LIN {X 0,Y 234.994,Z 198.991,A -85,B 0,C 180,E1 -19665.872,E2 -19665.872} C_VEL
LIN {X 0,Y 235.262,Z 200.964,A -85,B 0,C 180,E1 -19668.915,E2 -19668.915} C_VEL
LIN {X 0,Y 235.336,Z 202.53,A -85,B 0,C 180,E1 -19671.163,E2 -19671.163} C_VEL
LIN {X 0,Y 235.127,Z 205.559,A -85,B 0,C 180,E1 -19675.132,E2 -19675.132} C_VEL
LIN {X 0,Y 236.112,Z 208.531,A -85,B 0,C 180,E1 -19675.455,E2 -19675.455} C_VEL
LIN {X 0,Y 240.672,Z 220.482,A -85,B 0,C 180,E1 -19677.002,E2 -19677.002} C_VEL
LIN {X 0,Y 244.007,Z 232.021,A -85,B 0,C 180,E1 -19678.611,E2 -19678.611} C_VEL
LIN {X 0,Y 246.229,Z 243.079,A -85,B 0,C 180,E1 -19680.305,E2 -19680.305} C_VEL
LIN {X 0,Y 247.437,Z 253.06,A -85,B 0,C 180,E1 -19682.016,E2 -19682.016} C_VEL
LIN {X 0,Y 247.369,Z 256.03,A -85,B 0,C 180,E1 -19682.536,E2 -19682.536} C_VEL
LIN {X 0,Y 245.059,Z 266.116,A -85,B 0,C 180,E1 -19684.294,E2 -19684.294} C_VEL
LIN {X 0,Y 242.891,Z 274.497,A -85,B 0,C 180,E1 -19686.104,E2 -19686.104} C_VEL
LIN {X 0,Y 240.296,Z 283.569,A -85,B 0,C 180,E1 -19688.557,E2 -19688.557} C_VEL
LIN {X 0,Y 238.141,Z 290.868,A -85,B 0,C 180,E1 -19691.057,E2 -19691.057} C_VEL
LIN {X 0,Y 236.506,Z 296.707,A -85,B 0,C 180,E1 -19693.602,E2 -19693.602} C_VEL
LIN {X 0,Y 234.979,Z 301.307,A -85,B 0,C 180,E1 -19696.156,E2 -19696.156} C_VEL
LIN {X 0,Y 234.316,Z 303.742,A -85,B 0,C 180,E1 -19697.88,E2 -19697.88} C_VEL
LIN {X 0,Y 233.756,Z 305.721,A -85,B 0,C 180,E1 -19699.607,E2 -19699.607} C_VEL
LIN {X 0,Y 233.332,Z 307.288,A -85,B 0,C 180,E1 -19701.338,E2 -19701.338} C_VEL
LIN {X 0,Y 233.048,Z 308.446,A -85,B 0,C 180,E1 -19703.071,E2 -19703.071} C_VEL
LIN {X 0,Y 232.884,Z 309.166,A -85,B 0,C 180,E1 -19704.805,E2 -19704.805} C_VEL
LIN {X 0,Y 232.805,Z 309.463,A -85,B 0,C 180,E1 -19708.269,E2 -19708.269} C_VEL
LIN {X 0,Y 232.834,Z 309.041,A -85,B 0,C 180,E1 -19709.999,E2 -19709.999} C_VEL
LIN {X 0,Y 233.162,Z 306.944,A -85,B 0,C 180,E1 -19713.455,E2 -19713.455} C_VEL
LIN {X 0,Y 233.699,Z 304.308,A -85,B 0,C 180,E1 -19716.04,E2 -19716.04} C_VEL
LIN {X 0,Y 234.385,Z 300.675,A -85,B 0,C 180,E1 -19718.621,E2 -19718.621} C_VEL
LIN {X 0,Y 235.457,Z 295.934,A -85,B 0,C 180,E1 -19721.185,E2 -19721.185} C_VEL
LIN {X 0,Y 237.199,Z 288.834,A -85,B 0,C 180,E1 -19724.147,E2 -19724.147} C_VEL
LIN {X 0,Y 239.174,Z 281.069,A -85,B 0,C 180,E1 -19726.646,E2 -19726.646} C_VEL
LIN {X 0,Y 241.478,Z 271.375,A -85,B 0,C 180,E1 -19729.11,E2 -19729.11} C_VEL
LIN {X 0,Y 243.532,Z 261.323,A -85,B 0,C 180,E1 -19731.142,E2 -19731.142} C_VEL
LIN {X 0,Y 245.429,Z 252.166,A -85,B 0,C 180,E1 -19732.608,E2 -19732.608} C_VEL
LIN {X 0,Y 244.466,Z 242.609,A -85,B 0,C 180,E1 -19734.155,E2 -19734.155} C_VEL
LIN {X 0,Y 242.465,Z 231.247,A -85,B 0,C 180,E1 -19735.768,E2 -19735.768} C_VEL
LIN {X 0,Y 239.316,Z 219.271,A -85,B 0,C 180,E1 -19737.274,E2 -19737.274} C_VEL
LIN {X 0,Y 235.407,Z 207.747,A -85,B 0,C 180,E1 -19738.557,E2 -19738.557} C_VEL
LIN {X 0,Y 234.73,Z 205.201,A -85,B 0,C 180,E1 -19738.831,E2 -19738.831} C_VEL
LIN {X 0,Y 235.027,Z 201.864,A -85,B 0,C 180,E1 -19743.144,E2 -19743.144} C_VEL
LIN {X 0,Y 234.981,Z 199.25,A -85,B 0,C 180,E1 -19746.735,E2 -19746.735} C_VEL
LIN {X 0,Y 234.904,Z 198.228,A -85,B 0,C 180,E1 -19748.932,E2 -19748.932} C_VEL
LIN {X 0,Y 234.887,Z 198.229,A -85,B 0,C 180,E1 -19753.481,E2 -19753.481} C_VEL
LIN {X 0,Y 234.963,Z 198.217,A -85,B 0,C 180,E1 -19756.531,E2 -19756.531} C_VEL
LIN {X 0,Y 234.943,Z 198.222,A -85,B 0,C 180,E1 -19761.083,E2 -19761.083} C_VEL
LIN {X 0,Y 234.92,Z 198.222,A -85,B 0,C 180,E1 -19765.36,E2 -19765.36} C_VEL
LIN {X 0,Y 234.906,Z 198.223,A -85,B 0,C 180,E1 -19769.428,E2 -19769.428} C_VEL
LIN {X 0,Y 234.977,Z 198.214,A -85,B 0,C 180,E1 -19773.792,E2 -19773.792} C_VEL
LIN {X 0,Y 235.029,Z 198.172,A -85,B 0,C 180,E1 -19778.971,E2 -19778.971} C_VEL
LIN {X 0,Y 235.098,Z 198.194,A -85,B 0,C 180,E1 -19783.042,E2 -19783.042} C_VEL
LIN {X 0,Y 235.145,Z 198.189,A -85,B 0,C 180,E1 -19787.923,E2 -19787.923} C_VEL
LIN {X 0,Y 235.376,Z 198.162,A -85,B 0,C 180,E1 -19791.414,E2 -19791.414} C_VEL
LIN {X 0,Y 235.388,Z 198.163,A -85,B 0,C 180,E1 -19793.14,E2 -19793.14} C_VEL
LIN {X 0,Y 235.571,Z 198.14,A -85,B 0,C 180,E1 -19798.29,E2 -19798.29} C_VEL
LIN {X 0,Y 235.582,Z 198.14,A -85,B 0,C 180,E1 -19801.709,E2 -19801.709} C_VEL
LIN {X 0,Y 235.381,Z 198.163,A -85,B 0,C 180,E1 -19806.859,E2 -19806.859} C_VEL
LIN {X 0,Y 235.216,Z 198.185,A -85,B 0,C 180,E1 -19810.327,E2 -19810.327} C_VEL
LIN {X 0,Y 235.073,Z 198.205,A -85,B 0,C 180,E1 -19815.609,E2 -19815.609} C_VEL
LIN {X 0,Y 235.009,Z 198.213,A -85,B 0,C 180,E1 -19819.205,E2 -19819.205} C_VEL
LIN {X 0,Y 234.978,Z 198.217,A -85,B 0,C 180,E1 -19822.881,E2 -19822.881} C_VEL
LIN {X 0,Y 234.952,Z 198.219,A -85,B 0,C 180,E1 -19826.659,E2 -19826.659} C_VEL
LIN {X 0,Y 234.914,Z 198.21,A -85,B 0,C 180,E1 -19830.57,E2 -19830.57} C_VEL
LIN {X 0,Y 234.945,Z 198.221,A -85,B 0,C 180,E1 -19834.635,E2 -19834.635} C_VEL
LIN {X 0,Y 234.953,Z 198.219,A -85,B 0,C 180,E1 -19838.955,E2 -19838.955} C_VEL
LIN {X 0,Y 234.997,Z 198.271,A -85,B 0,C 180,E1 -19840.295,E2 -19840.295} C_VEL
LIN {X 0,Y 235.555,Z 201.483,A -85,B 0,C 180,E1 -19844.276,E2 -19844.276} C_VEL
LIN {X 0,Y 236.061,Z 204.807,A -85,B 0,C 180,E1 -19848.099,E2 -19848.099} C_VEL
LIN {X 0,Y 236.491,Z 207.822,A -85,B 0,C 180,E1 -19851.391,E2 -19851.391} C_VEL
LIN {X 0,Y 236.489,Z 209.071,A -85,B 0,C 180,E1 -19852.68,E2 -19852.68} C_VEL
LIN {X 0,Y 235.807,Z 210.061,A -85,B 0,C 180,E1 -19853.591,E2 -19853.591} C_VEL
LIN {X 0,Y 232.815,Z 211.85,A -85,B 0,C 180,E1 -19854.992,E2 -19854.992} C_VEL
LIN {X 0,Y 229.663,Z 213.67,A -85,B 0,C 180,E1 -19856.422,E2 -19856.422} C_VEL
LIN {X 0,Y 228.79,Z 214.713,A -85,B 0,C 180,E1 -19857.371,E2 -19857.371} C_VEL
LIN {X 0,Y 228.579,Z 215.69,A -85,B 0,C 180,E1 -19858.329,E2 -19858.329} C_VEL
LIN {X 0,Y 232.328,Z 229.691,A -85,B 0,C 180,E1 -19859.748,E2 -19859.748} C_VEL
LIN {X 0,Y 234.878,Z 242.527,A -85,B 0,C 180,E1 -19861.279,E2 -19861.279} C_VEL
LIN {X 0,Y 236.253,Z 254.477,A -85,B 0,C 180,E1 -19862.92,E2 -19862.92} C_VEL
LIN {X 0,Y 236.687,Z 265.741,A -85,B 0,C 180,E1 -19864.736,E2 -19864.736} C_VEL
LIN {X 0,Y 236.561,Z 270.846,A -85,B 0,C 180,E1 -19865.659,E2 -19865.659} C_VEL
LIN {X 0,Y 234.302,Z 280.591,A -85,B 0,C 180,E1 -19867.518,E2 -19867.518} C_VEL
LIN {X 0,Y 232.039,Z 290.368,A -85,B 0,C 180,E1 -19869.872,E2 -19869.872} C_VEL
LIN {X 0,Y 230.139,Z 298.132,A -85,B 0,C 180,E1 -19872.221,E2 -19872.221} C_VEL
LIN {X 0,Y 228.441,Z 305.049,A -85,B 0,C 180,E1 -19874.843,E2 -19874.843} C_VEL
LIN {X 0,Y 227.127,Z 310.591,A -85,B 0,C 180,E1 -19877.493,E2 -19877.493} C_VEL
LIN {X 0,Y 226.317,Z 314.942,A -85,B 0,C 180,E1 -19880.168,E2 -19880.168} C_VEL
LIN {X 0,Y 225.82,Z 318.217,A -85,B 0,C 180,E1 -19882.851,E2 -19882.851} C_VEL
LIN {X 0,Y 225.589,Z 320.491,A -85,B 0,C 180,E1 -19885.508,E2 -19885.508} C_VEL
LIN {X 0,Y 225.643,Z 321.872,A -85,B 0,C 180,E1 -19888.216,E2 -19888.216} C_VEL
LIN {X 0,Y 225.714,Z 322.254,A -85,B 0,C 180,E1 -19890.001,E2 -19890.001} C_VEL
LIN {X 0,Y 225.636,Z 322.245,A -85,B 0,C 180,E1 -19891.786,E2 -19891.786} C_VEL
LIN {X 0,Y 225.585,Z 321.472,A -85,B 0,C 180,E1 -19894.48,E2 -19894.48} C_VEL
LIN {X 0,Y 225.822,Z 319.809,A -85,B 0,C 180,E1 -19897.152,E2 -19897.152} C_VEL
LIN {X 0,Y 226.356,Z 317.2,A -85,B 0,C 180,E1 -19899.833,E2 -19899.833} C_VEL
LIN {X 0,Y 227.26,Z 313.584,A -85,B 0,C 180,E1 -19902.502,E2 -19902.502} C_VEL
LIN {X 0,Y 228.572,Z 308.866,A -85,B 0,C 180,E1 -19905.15,E2 -19905.15} C_VEL
LIN {X 0,Y 230.423,Z 302.906,A -85,B 0,C 180,E1 -19907.758,E2 -19907.758} C_VEL
LIN {X 0,Y 232.584,Z 295.571,A -85,B 0,C 180,E1 -19910.305,E2 -19910.305} C_VEL
LIN {X 0,Y 234.7,Z 287.935,A -85,B 0,C 180,E1 -19912.444,E2 -19912.444} C_VEL
LIN {X 0,Y 237.272,Z 278.802,A -85,B 0,C 180,E1 -19914.499,E2 -19914.499} C_VEL
LIN {X 0,Y 238.862,Z 272.268,A -85,B 0,C 180,E1 -19915.72,E2 -19915.72} C_VEL
LIN {X 0,Y 238.703,Z 261.301,A -85,B 0,C 180,E1 -19917.736,E2 -19917.736} C_VEL
LIN {X 0,Y 237.746,Z 250.445,A -85,B 0,C 180,E1 -19919.471,E2 -19919.471} C_VEL
LIN {X 0,Y 235.848,Z 239.193,A -85,B 0,C 180,E1 -19921.074,E2 -19921.074} C_VEL
LIN {X 0,Y 232.84,Z 226.637,A -85,B 0,C 180,E1 -19922.652,E2 -19922.652} C_VEL
LIN {X 0,Y 229.491,Z 216.356,A -85,B 0,C 180,E1 -19923.854,E2 -19923.854} C_VEL
LIN {X 0,Y 229.383,Z 215.464,A -85,B 0,C 180,E1 -19923.937,E2 -19923.937} C_VEL
LIN {X 0,Y 229.656,Z 213.876,A -85,B 0,C 180,E1 -19925.551,E2 -19925.551} C_VEL
LIN {X 0,Y 229.77,Z 210.838,A -85,B 0,C 180,E1 -19928.83,E2 -19928.83} C_VEL
LIN {X 0,Y 229.352,Z 207.534,A -85,B 0,C 180,E1 -19932.657,E2 -19932.657} C_VEL
LIN {X 0,Y 228.983,Z 205.536,A -85,B 0,C 180,E1 -19935.096,E2 -19935.096} C_VEL
LIN {X 0,Y 228.349,Z 202.015,A -85,B 0,C 180,E1 -19939.735,E2 -19939.735} C_VEL
LIN {X 0,Y 227.903,Z 199.162,A -85,B 0,C 180,E1 -19943.813,E2 -19943.813} C_VEL
LIN {X 0,Y 227.848,Z 199.108,A -85,B 0,C 180,E1 -19948.375,E2 -19948.375} C_VEL
LIN {X 0,Y 227.86,Z 199.103,A -85,B 0,C 180,E1 -19952.442,E2 -19952.442} C_VEL
LIN {X 0,Y 227.924,Z 199.094,A -85,B 0,C 180,E1 -19956.369,E2 -19956.369} C_VEL
LIN {X 0,Y 227.957,Z 199.09,A -85,B 0,C 180,E1 -19960.176,E2 -19960.176} C_VEL
LIN {X 0,Y 228.052,Z 199.077,A -85,B 0,C 180,E1 -19963.898,E2 -19963.898} C_VEL
LIN {X 0,Y 228.058,Z 199.075,A -85,B 0,C 180,E1 -19967.543,E2 -19967.543} C_VEL
LIN {X 0,Y 228.255,Z 199.052,A -85,B 0,C 180,E1 -19971.144,E2 -19971.144} C_VEL
LIN {X 0,Y 228.311,Z 199.046,A -85,B 0,C 180,E1 -19972.928,E2 -19972.928} C_VEL
LIN {X 0,Y 228.538,Z 199.017,A -85,B 0,C 180,E1 -19978.238,E2 -19978.238} C_VEL
LIN {X 0,Y 228.551,Z 199.015,A -85,B 0,C 180,E1 -19981.763,E2 -19981.763} C_VEL
LIN {X 0,Y 228.308,Z 199.044,A -85,B 0,C 180,E1 -19987.073,E2 -19987.073} C_VEL
LIN {X 0,Y 228.13,Z 199.067,A -85,B 0,C 180,E1 -19990.652,E2 -19990.652} C_VEL
LIN {X 0,Y 228.04,Z 199.079,A -85,B 0,C 180,E1 -19996.104,E2 -19996.104} C_VEL
LIN {X 0,Y 227.931,Z 199.093,A -85,B 0,C 180,E1 -19999.827,E2 -19999.827} C_VEL
LIN {X 0,Y 227.904,Z 199.096,A -85,B 0,C 180,E1 -20003.634,E2 -20003.634} C_VEL
LIN {X 0,Y 227.871,Z 199.101,A -85,B 0,C 180,E1 -20007.558,E2 -20007.558} C_VEL
LIN {X 0,Y 227.859,Z 199.102,A -85,B 0,C 180,E1 -20011.625,E2 -20011.625} C_VEL
LIN {X 0,Y 227.875,Z 199.1,A -85,B 0,C 180,E1 -20015.874,E2 -20015.874} C_VEL
LIN {X 0,Y 227.82,Z 199.106,A -85,B 0,C 180,E1 -20020.379,E2 -20020.379} C_VEL
LIN {X 0,Y 227.8,Z 199.111,A -85,B 0,C 180,E1 -20022.746,E2 -20022.746} C_VEL
LIN {X 0,Y 227.93,Z 199.817,A -85,B 0,C 180,E1 -20025.169,E2 -20025.169} C_VEL
LIN {X 0,Y 228.262,Z 202.698,A -85,B 0,C 180,E1 -20029.718,E2 -20029.718} C_VEL
LIN {X 0,Y 228.207,Z 205.665,A -85,B 0,C 180,E1 -20033.954,E2 -20033.954} C_VEL
LIN {X 0,Y 229.317,Z 208.854,A -85,B 0,C 180,E1 -20034.329,E2 -20034.329} C_VEL
LIN {X 0,Y 233.879,Z 220.739,A -85,B 0,C 180,E1 -20035.961,E2 -20035.961} C_VEL
LIN {X 0,Y 236.893,Z 230.669,A -85,B 0,C 180,E1 -20037.423,E2 -20037.423} C_VEL
LIN {X 0,Y 239.325,Z 241.897,A -85,B 0,C 180,E1 -20039.201,E2 -20039.201} C_VEL
LIN {X 0,Y 240.688,Z 251.922,A -85,B 0,C 180,E1 -20040.963,E2 -20040.963} C_VEL
LIN {X 0,Y 240.842,Z 257.166,A -85,B 0,C 180,E1 -20041.934,E2 -20041.934} C_VEL
LIN {X 0,Y 238.38,Z 267.157,A -85,B 0,C 180,E1 -20043.754,E2 -20043.754} C_VEL
LIN {X 0,Y 235.922,Z 276.204,A -85,B 0,C 180,E1 -20045.821,E2 -20045.821} C_VEL
LIN {X 0,Y 233.255,Z 285.017,A -85,B 0,C 180,E1 -20048.341,E2 -20048.341} C_VEL
LIN {X 0,Y 231.074,Z 292.072,A -85,B 0,C 180,E1 -20050.916,E2 -20050.916} C_VEL
LIN {X 0,Y 229.676,Z 296.838,A -85,B 0,C 180,E1 -20053.1,E2 -20053.1} C_VEL
LIN {X 0,Y 228.059,Z 301.452,A -85,B 0,C 180,E1 -20055.727,E2 -20055.727} C_VEL
LIN {X 0,Y 227.355,Z 303.901,A -85,B 0,C 180,E1 -20057.503,E2 -20057.503} C_VEL
LIN {X 0,Y 226.758,Z 305.886,A -85,B 0,C 180,E1 -20059.282,E2 -20059.282} C_VEL
LIN {X 0,Y 226.293,Z 307.46,A -85,B 0,C 180,E1 -20061.066,E2 -20061.066} C_VEL
LIN {X 0,Y 225.996,Z 308.626,A -85,B 0,C 180,E1 -20062.854,E2 -20062.854} C_VEL
LIN {X 0,Y 225.768,Z 309.442,A -85,B 0,C 180,E1 -20064.972,E2 -20064.972} C_VEL
LIN {X 0,Y 225.72,Z 309.664,A -85,B 0,C 180,E1 -20068.215,E2 -20068.215} C_VEL
LIN {X 0,Y 225.747,Z 309.25,A -85,B 0,C 180,E1 -20069.999,E2 -20069.999} C_VEL
LIN {X 0,Y 225.853,Z 308.408,A -85,B 0,C 180,E1 -20071.782,E2 -20071.782} C_VEL
LIN {X 0,Y 226.09,Z 307.168,A -85,B 0,C 180,E1 -20073.563,E2 -20073.563} C_VEL
LIN {X 0,Y 226.634,Z 304.545,A -85,B 0,C 180,E1 -20076.229,E2 -20076.229} C_VEL
LIN {X 0,Y 227.379,Z 300.925,A -85,B 0,C 180,E1 -20078.888,E2 -20078.888} C_VEL
LIN {X 0,Y 228.519,Z 296.198,A -85,B 0,C 180,E1 -20081.529,E2 -20081.529} C_VEL
LIN {X 0,Y 230.331,Z 289.114,A -85,B 0,C 180,E1 -20084.578,E2 -20084.578} C_VEL
LIN {X 0,Y 232.401,Z 281.376,A -85,B 0,C 180,E1 -20087.146,E2 -20087.146} C_VEL
LIN {X 0,Y 234.778,Z 271.705,A -85,B 0,C 180,E1 -20089.677,E2 -20089.677} C_VEL
LIN {X 0,Y 236.948,Z 261.692,A -85,B 0,C 180,E1 -20091.759,E2 -20091.759} C_VEL
LIN {X 0,Y 238.789,Z 253.116,A -85,B 0,C 180,E1 -20093.18,E2 -20093.18} C_VEL
LIN {X 0,Y 237.942,Z 244.186,A -85,B 0,C 180,E1 -20094.695,E2 -20094.695} C_VEL
LIN {X 0,Y 236.166,Z 233.622,A -85,B 0,C 180,E1 -20096.299,E2 -20096.299} C_VEL
LIN {X 0,Y 233.467,Z 222.697,A -85,B 0,C 180,E1 -20097.782,E2 -20097.782} C_VEL
LIN {X 0,Y 229.335,Z 210.086,A -85,B 0,C 180,E1 -20099.303,E2 -20099.303} C_VEL
LIN {X 0,Y 227.736,Z 205.422,A -85,B 0,C 180,E1 -20099.839,E2 -20099.839} C_VEL
LIN {X 0,Y 228.003,Z 202.525,A -85,B 0,C 180,E1 -20103.695,E2 -20103.695} C_VEL
LIN {X 0,Y 227.982,Z 200.413,A -85,B 0,C 180,E1 -20106.725,E2 -20106.725} C_VEL
LIN {X 0,Y 227.856,Z 199.502,A -85,B 0,C 180,E1 -20108.084,E2 -20108.084} C_VEL
LIN {X 0,Y 227.811,Z 199.109,A -85,B 0,C 180,E1 -20110.375,E2 -20110.375} C_VEL
LIN {X 0,Y 227.85,Z 199.103,A -85,B 0,C 180,E1 -20115.183,E2 -20115.183} C_VEL
LIN {X 0,Y 227.906,Z 199.097,A -85,B 0,C 180,E1 -20117.733,E2 -20117.733} C_VEL
LIN {X 0,Y 227.856,Z 199.101,A -85,B 0,C 180,E1 -20121.91,E2 -20121.91} C_VEL
LIN {X 0,Y 227.866,Z 199.101,A -85,B 0,C 180,E1 -20126.374,E2 -20126.374} C_VEL
LIN {X 0,Y 227.888,Z 199.098,A -85,B 0,C 180,E1 -20130.433,E2 -20130.433} C_VEL
LIN {X 0,Y 227.914,Z 199.093,A -85,B 0,C 180,E1 -20134.423,E2 -20134.423} C_VEL
LIN {X 0,Y 227.99,Z 199.05,A -85,B 0,C 180,E1 -20138.289,E2 -20138.289} C_VEL
LIN {X 0,Y 228.026,Z 199.071,A -85,B 0,C 180,E1 -20142.816,E2 -20142.816} C_VEL
LIN {X 0,Y 228.086,Z 199.071,A -85,B 0,C 180,E1 -20147.543,E2 -20147.543} C_VEL
LIN {X 0,Y 228.314,Z 199.041,A -85,B 0,C 180,E1 -20151.146,E2 -20151.146} C_VEL
LIN {X 0,Y 228.341,Z 199.04,A -85,B 0,C 180,E1 -20152.928,E2 -20152.928} C_VEL
LIN {X 0,Y 228.53,Z 199.017,A -85,B 0,C 180,E1 -20158.237,E2 -20158.237} C_VEL
LIN {X 0,Y 228.542,Z 199.017,A -85,B 0,C 180,E1 -20161.762,E2 -20161.762} C_VEL
LIN {X 0,Y 228.332,Z 199.042,A -85,B 0,C 180,E1 -20167.072,E2 -20167.072} C_VEL
LIN {X 0,Y 228.137,Z 199.067,A -85,B 0,C 180,E1 -20170.651,E2 -20170.651} C_VEL
LIN {X 0,Y 228.024,Z 199.081,A -85,B 0,C 180,E1 -20176.104,E2 -20176.104} C_VEL
LIN {X 0,Y 227.947,Z 199.092,A -85,B 0,C 180,E1 -20179.825,E2 -20179.825} C_VEL
LIN {X 0,Y 227.916,Z 199.095,A -85,B 0,C 180,E1 -20183.632,E2 -20183.632} C_VEL
LIN {X 0,Y 227.868,Z 199.1,A -85,B 0,C 180,E1 -20187.557,E2 -20187.557} C_VEL
LIN {X 0,Y 227.856,Z 199.092,A -85,B 0,C 180,E1 -20191.624,E2 -20191.624} C_VEL
LIN {X 0,Y 227.886,Z 199.099,A -85,B 0,C 180,E1 -20195.871,E2 -20195.871} C_VEL
LIN {X 0,Y 227.988,Z 199.297,A -85,B 0,C 180,E1 -20199.876,E2 -20199.876} C_VEL
LIN {X 0,Y 228.357,Z 201.395,A -85,B 0,C 180,E1 -20202.616,E2 -20202.616} C_VEL
LIN {X 0,Y 228.977,Z 205.386,A -85,B 0,C 180,E1 -20207.445,E2 -20207.445} C_VEL
LIN {X 0,Y 229.444,Z 208.657,A -85,B 0,C 180,E1 -20211.143,E2 -20211.143} C_VEL
LIN {X 0,Y 229.38,Z 211.736,A -85,B 0,C 180,E1 -20214.403,E2 -20214.403} C_VEL
LIN {X 0,Y 228.79,Z 214.713,A -85,B 0,C 180,E1 -20217.371,E2 -20217.371} C_VEL
LIN {X 0,Y 229.046,Z 215.928,A -85,B 0,C 180,E1 -20218.009,E2 -20218.009} C_VEL
LIN {X 0,Y 230.107,Z 218.575,A -85,B 0,C 180,E1 -20218.663,E2 -20218.663} C_VEL
LIN {X 0,Y 231.77,Z 222.871,A -85,B 0,C 180,E1 -20219.187,E2 -20219.187} C_VEL
LIN {X 0,Y 232.069,Z 226.734,A -85,B 0,C 180,E1 -20219.491,E2 -20219.491} C_VEL
LIN {X 0,Y 231.275,Z 231.15,A -85,B 0,C 180,E1 -20219.698,E2 -20219.698} C_VEL
LIN {X 0,Y 228.54,Z 239.929,A -85,B 0,C 180,E1 -20220.171,E2 -20220.171} C_VEL
LIN {X 0,Y 228.37,Z 243.73,A -85,B 0,C 180,E1 -20220.571,E2 -20220.571} C_VEL
LIN {X 0,Y 229.614,Z 254.399,A -85,B 0,C 180,E1 -20222.121,E2 -20222.121} C_VEL
LIN {X 0,Y 229.988,Z 265.661,A -85,B 0,C 180,E1 -20224.002,E2 -20224.002} C_VEL
LIN {X 0,Y 229.823,Z 271.676,A -85,B 0,C 180,E1 -20225.139,E2 -20225.139} C_VEL
LIN {X 0,Y 227.265,Z 282.226,A -85,B 0,C 180,E1 -20227.263,E2 -20227.263} C_VEL
LIN {X 0,Y 225.196,Z 290.719,A -85,B 0,C 180,E1 -20229.431,E2 -20229.431} C_VEL
LIN {X 0,Y 223.37,Z 297.855,A -85,B 0,C 180,E1 -20231.664,E2 -20231.664} C_VEL
LIN {X 0,Y 221.57,Z 304.786,A -85,B 0,C 180,E1 -20234.361,E2 -20234.361} C_VEL
LIN {X 0,Y 220.144,Z 310.34,A -85,B 0,C 180,E1 -20237.089,E2 -20237.089} C_VEL
LIN {X 0,Y 219.301,Z 314.704,A -85,B 0,C 180,E1 -20239.85,E2 -20239.85} C_VEL
LIN {X 0,Y 218.759,Z 317.99,A -85,B 0,C 180,E1 -20242.618,E2 -20242.618} C_VEL
LIN {X 0,Y 218.486,Z 320.475,A -85,B 0,C 180,E1 -20245.688,E2 -20245.688} C_VEL
LIN {X 0,Y 218.541,Z 321.666,A -85,B 0,C 180,E1 -20248.159,E2 -20248.159} C_VEL
LIN {X 0,Y 218.629,Z 322.054,A -85,B 0,C 180,E1 -20250.001,E2 -20250.001} C_VEL
LIN {X 0,Y 218.534,Z 322.05,A -85,B 0,C 180,E1 -20251.844,E2 -20251.844} C_VEL
LIN {X 0,Y 218.482,Z 321.432,A -85,B 0,C 180,E1 -20254.297,E2 -20254.297} C_VEL
LIN {X 0,Y 218.761,Z 319.634,A -85,B 0,C 180,E1 -20257.384,E2 -20257.384} C_VEL
LIN {X 0,Y 219.339,Z 317.036,A -85,B 0,C 180,E1 -20260.151,E2 -20260.151} C_VEL
LIN {X 0,Y 220.28,Z 313.43,A -85,B 0,C 180,E1 -20262.905,E2 -20262.905} C_VEL
LIN {X 0,Y 221.71,Z 308.725,A -85,B 0,C 180,E1 -20265.631,E2 -20265.631} C_VEL
LIN {X 0,Y 223.625,Z 302.778,A -85,B 0,C 180,E1 -20268.317,E2 -20268.317} C_VEL
LIN {X 0,Y 225.731,Z 296.057,A -85,B 0,C 180,E1 -20270.74,E2 -20270.74} C_VEL
LIN {X 0,Y 228.14,Z 287.841,A -85,B 0,C 180,E1 -20273.127,E2 -20273.127} C_VEL
LIN {X 0,Y 230.805,Z 278.729,A -85,B 0,C 180,E1 -20275.232,E2 -20275.232} C_VEL
LIN {X 0,Y 232.227,Z 273.395,A -85,B 0,C 180,E1 -20276.269,E2 -20276.269} C_VEL
LIN {X 0,Y 232.173,Z 262.42,A -85,B 0,C 180,E1 -20278.39,E2 -20278.39} C_VEL
LIN {X 0,Y 231.295,Z 251.376,A -85,B 0,C 180,E1 -20280.249,E2 -20280.249} C_VEL
LIN {X 0,Y 229.514,Z 240.364,A -85,B 0,C 180,E1 -20281.909,E2 -20281.909} C_VEL
LIN {X 0,Y 226.778,Z 228.584,A -85,B 0,C 180,E1 -20283.505,E2 -20283.505} C_VEL
LIN {X 0,Y 223.252,Z 217.971,A -85,B 0,C 180,E1 -20284.868,E2 -20284.868} C_VEL
LIN {X 0,Y 222.543,Z 215.254,A -85,B 0,C 180,E1 -20285.168,E2 -20285.168} C_VEL
LIN {X 0,Y 222.723,Z 212.757,A -85,B 0,C 180,E1 -20287.92,E2 -20287.92} C_VEL
LIN {X 0,Y 222.441,Z 209.617,A -85,B 0,C 180,E1 -20291.565,E2 -20291.565} C_VEL
LIN {X 0,Y 221.879,Z 206.253,A -85,B 0,C 180,E1 -20295.825,E2 -20295.825} C_VEL
LIN {X 0,Y 221.304,Z 202.796,A -85,B 0,C 180,E1 -20300.57,E2 -20300.57} C_VEL
LIN {X 0,Y 220.812,Z 199.984,A -85,B 0,C 180,E1 -20304.908,E2 -20304.908} C_VEL
LIN {X 0,Y 220.826,Z 199.982,A -85,B 0,C 180,E1 -20309.389,E2 -20309.389} C_VEL
LIN {X 0,Y 220.884,Z 199.971,A -85,B 0,C 180,E1 -20313.548,E2 -20313.548} C_VEL
LIN {X 0,Y 220.93,Z 199.965,A -85,B 0,C 180,E1 -20317.559,E2 -20317.559} C_VEL
LIN {X 0,Y 220.982,Z 199.96,A -85,B 0,C 180,E1 -20322.565,E2 -20322.565} C_VEL
LIN {X 0,Y 220.998,Z 199.956,A -85,B 0,C 180,E1 -20327.138,E2 -20327.138} C_VEL
LIN {X 0,Y 221.193,Z 199.933,A -85,B 0,C 180,E1 -20330.859,E2 -20330.859} C_VEL
LIN {X 0,Y 221.247,Z 199.925,A -85,B 0,C 180,E1 -20332.701,E2 -20332.701} C_VEL
LIN {X 0,Y 221.496,Z 199.894,A -85,B 0,C 180,E1 -20338.182,E2 -20338.182} C_VEL
LIN {X 0,Y 221.509,Z 199.893,A -85,B 0,C 180,E1 -20341.819,E2 -20341.819} C_VEL
LIN {X 0,Y 221.242,Z 199.925,A -85,B 0,C 180,E1 -20347.3,E2 -20347.3} C_VEL
LIN {X 0,Y 221.051,Z 199.949,A -85,B 0,C 180,E1 -20350.998,E2 -20350.998} C_VEL
LIN {X 0,Y 221.003,Z 199.955,A -85,B 0,C 180,E1 -20356.631,E2 -20356.631} C_VEL
LIN {X 0,Y 220.882,Z 199.97,A -85,B 0,C 180,E1 -20360.488,E2 -20360.488} C_VEL
LIN {X 0,Y 220.858,Z 199.972,A -85,B 0,C 180,E1 -20364.437,E2 -20364.437} C_VEL
LIN {X 0,Y 220.819,Z 199.978,A -85,B 0,C 180,E1 -20368.517,E2 -20368.517} C_VEL
LIN {X 0,Y 220.81,Z 199.981,A -85,B 0,C 180,E1 -20372.758,E2 -20372.758} C_VEL
LIN {X 0,Y 220.804,Z 199.978,A -85,B 0,C 180,E1 -20377.279,E2 -20377.279} C_VEL
LIN {X 0,Y 220.789,Z 199.981,A -85,B 0,C 180,E1 -20380.189,E2 -20380.189} C_VEL
LIN {X 0,Y 220.759,Z 199.987,A -85,B 0,C 180,E1 -20382.93,E2 -20382.93} C_VEL
LIN {X 0,Y 221.061,Z 202.193,A -85,B 0,C 180,E1 -20386.99,E2 -20386.99} C_VEL
LIN {X 0,Y 221.276,Z 204.455,A -85,B 0,C 180,E1 -20390.565,E2 -20390.565} C_VEL
LIN {X 0,Y 221.257,Z 206.079,A -85,B 0,C 180,E1 -20392.691,E2 -20392.691} C_VEL
LIN {X 0,Y 222.417,Z 209.19,A -85,B 0,C 180,E1 -20393.098,E2 -20393.098} C_VEL
LIN {X 0,Y 224.554,Z 214.034,A -85,B 0,C 180,E1 -20393.821,E2 -20393.821} C_VEL
LIN {X 0,Y 228.576,Z 225.286,A -85,B 0,C 180,E1 -20395.514,E2 -20395.514} C_VEL
LIN {X 0,Y 231.581,Z 236.568,A -85,B 0,C 180,E1 -20397.319,E2 -20397.319} C_VEL
LIN {X 0,Y 233.558,Z 247.534,A -85,B 0,C 180,E1 -20399.234,E2 -20399.234} C_VEL
LIN {X 0,Y 234.415,Z 257.086,A -85,B 0,C 180,E1 -20401.076,E2 -20401.076} C_VEL
LIN {X 0,Y 232.327,Z 266.203,A -85,B 0,C 180,E1 -20402.772,E2 -20402.772} C_VEL
LIN {X 0,Y 229.923,Z 274.64,A -85,B 0,C 180,E1 -20404.664,E2 -20404.664} C_VEL
LIN {X 0,Y 227.071,Z 283.765,A -85,B 0,C 180,E1 -20407.24,E2 -20407.24} C_VEL
LIN {X 0,Y 224.454,Z 291.807,A -85,B 0,C 180,E1 -20410.157,E2 -20410.157} C_VEL
LIN {X 0,Y 222.86,Z 296.97,A -85,B 0,C 180,E1 -20412.567,E2 -20412.567} C_VEL
LIN {X 0,Y 221.154,Z 301.598,A -85,B 0,C 180,E1 -20415.272,E2 -20415.272} C_VEL
LIN {X 0,Y 220.407,Z 304.059,A -85,B 0,C 180,E1 -20417.102,E2 -20417.102} C_VEL
LIN {X 0,Y 219.761,Z 306.052,A -85,B 0,C 180,E1 -20418.937,E2 -20418.937} C_VEL
LIN {X 0,Y 219.274,Z 307.631,A -85,B 0,C 180,E1 -20420.778,E2 -20420.778} C_VEL
LIN {X 0,Y 218.94,Z 308.807,A -85,B 0,C 180,E1 -20422.622,E2 -20422.622} C_VEL
LIN {X 0,Y 218.671,Z 309.705,A -85,B 0,C 180,E1 -20425.099,E2 -20425.099} C_VEL
LIN {X 0,Y 218.636,Z 309.864,A -85,B 0,C 180,E1 -20428.157,E2 -20428.157} C_VEL
LIN {X 0,Y 218.661,Z 309.458,A -85,B 0,C 180,E1 -20429.999,E2 -20429.999} C_VEL
LIN {X 0,Y 218.772,Z 308.626,A -85,B 0,C 180,E1 -20431.84,E2 -20431.84} C_VEL
LIN {X 0,Y 219.021,Z 307.392,A -85,B 0,C 180,E1 -20433.678,E2 -20433.678} C_VEL
LIN {X 0,Y 219.646,Z 304.372,A -85,B 0,C 180,E1 -20436.788,E2 -20436.788} C_VEL
LIN {X 0,Y 220.734,Z 299.757,A -85,B 0,C 180,E1 -20440.083,E2 -20440.083} C_VEL
LIN {X 0,Y 222.294,Z 293.651,A -85,B 0,C 180,E1 -20443.249,E2 -20443.249} C_VEL
LIN {X 0,Y 224.165,Z 286.991,A -85,B 0,C 180,E1 -20445.92,E2 -20445.92} C_VEL
LIN {X 0,Y 226.417,Z 278.727,A -85,B 0,C 180,E1 -20448.549,E2 -20448.549} C_VEL
LIN {X 0,Y 228.56,Z 270.219,A -85,B 0,C 180,E1 -20450.706,E2 -20450.706} C_VEL
LIN {X 0,Y 230.851,Z 259.73,A -85,B 0,C 180,E1 -20452.837,E2 -20452.837} C_VEL
LIN {X 0,Y 231.987,Z 254.912,A -85,B 0,C 180,E1 -20453.641,E2 -20453.641} C_VEL
LIN {X 0,Y 231.699,Z 248.424,A -85,B 0,C 180,E1 -20454.813,E2 -20454.813} C_VEL
LIN {X 0,Y 230.071,Z 237.139,A -85,B 0,C 180,E1 -20456.67,E2 -20456.67} C_VEL
LIN {X 0,Y 227.675,Z 226.489,A -85,B 0,C 180,E1 -20458.233,E2 -20458.233} C_VEL
LIN {X 0,Y 223.88,Z 214.142,A -85,B 0,C 180,E1 -20459.865,E2 -20459.865} C_VEL
LIN {X 0,Y 220.848,Z 206.204,A -85,B 0,C 180,E1 -20460.843,E2 -20460.843} C_VEL
LIN {X 0,Y 220.774,Z 205.648,A -85,B 0,C 180,E1 -20460.896,E2 -20460.896} C_VEL
LIN {X 0,Y 220.974,Z 202.791,A -85,B 0,C 180,E1 -20464.919,E2 -20464.919} C_VEL
LIN {X 0,Y 220.916,Z 201.176,A -85,B 0,C 180,E1 -20467.313,E2 -20467.313} C_VEL
LIN {X 0,Y 220.78,Z 199.985,A -85,B 0,C 180,E1 -20469.538,E2 -20469.538} C_VEL
LIN {X 0,Y 220.78,Z 199.986,A -85,B 0,C 180,E1 -20474.447,E2 -20474.447} C_VEL
LIN {X 0,Y 220.849,Z 199.975,A -85,B 0,C 180,E1 -20478.065,E2 -20478.065} C_VEL
LIN {X 0,Y 220.827,Z 199.978,A -85,B 0,C 180,E1 -20482.709,E2 -20482.709} C_VEL
LIN {X 0,Y 220.802,Z 199.979,A -85,B 0,C 180,E1 -20487.241,E2 -20487.241} C_VEL
LIN {X 0,Y 220.811,Z 199.977,A -85,B 0,C 180,E1 -20491.482,E2 -20491.482} C_VEL
LIN {X 0,Y 220.861,Z 199.965,A -85,B 0,C 180,E1 -20495.564,E2 -20495.564} C_VEL
LIN {X 0,Y 220.905,Z 199.928,A -85,B 0,C 180,E1 -20499.515,E2 -20499.515} C_VEL
LIN {X 0,Y 221.005,Z 199.949,A -85,B 0,C 180,E1 -20503.369,E2 -20503.369} C_VEL
LIN {X 0,Y 221.113,Z 199.93,A -85,B 0,C 180,E1 -20509.005,E2 -20509.005} C_VEL
LIN {X 0,Y 221.295,Z 199.919,A -85,B 0,C 180,E1 -20512.701,E2 -20512.701} C_VEL
LIN {X 0,Y 221.488,Z 199.892,A -85,B 0,C 180,E1 -20518.181,E2 -20518.181} C_VEL
LIN {X 0,Y 221.5,Z 199.895,A -85,B 0,C 180,E1 -20521.818,E2 -20521.818} C_VEL
LIN {X 0,Y 221.267,Z 199.923,A -85,B 0,C 180,E1 -20527.299,E2 -20527.299} C_VEL
LIN {X 0,Y 221.085,Z 199.947,A -85,B 0,C 180,E1 -20530.995,E2 -20530.995} C_VEL
LIN {X 0,Y 220.989,Z 199.958,A -85,B 0,C 180,E1 -20536.632,E2 -20536.632} C_VEL
LIN {X 0,Y 220.903,Z 199.969,A -85,B 0,C 180,E1 -20540.485,E2 -20540.485} C_VEL
LIN {X 0,Y 220.86,Z 199.974,A -85,B 0,C 180,E1 -20544.435,E2 -20544.435} C_VEL
LIN {X 0,Y 220.819,Z 199.976,A -85,B 0,C 180,E1 -20548.516,E2 -20548.516} C_VEL
LIN {X 0,Y 220.808,Z 199.978,A -85,B 0,C 180,E1 -20552.757,E2 -20552.757} C_VEL
LIN {X 0,Y 220.825,Z 199.979,A -85,B 0,C 180,E1 -20557.29,E2 -20557.29} C_VEL
LIN {X 0,Y 220.858,Z 199.975,A -85,B 0,C 180,E1 -20558.937,E2 -20558.937} C_VEL
LIN {X 0,Y 221.401,Z 203.068,A -85,B 0,C 180,E1 -20563.112,E2 -20563.112} C_VEL
LIN {X 0,Y 221.872,Z 205.969,A -85,B 0,C 180,E1 -20566.765,E2 -20566.765} C_VEL
LIN {X 0,Y 222.376,Z 209.405,A -85,B 0,C 180,E1 -20570.801,E2 -20570.801} C_VEL
LIN {X 0,Y 222.361,Z 212.519,A -85,B 0,C 180,E1 -20574.222,E2 -20574.222} C_VEL
LIN {X 0,Y 221.76,Z 215.507,A -85,B 0,C 180,E1 -20577.273,E2 -20577.273} C_VEL
LIN {X 0,Y 222.584,Z 218.658,A -85,B 0,C 180,E1 -20577.587,E2 -20577.587} C_VEL
LIN {X 0,Y 226.03,Z 231.421,A -85,B 0,C 180,E1 -20579.009,E2 -20579.009} C_VEL
LIN {X 0,Y 228.37,Z 243.73,A -85,B 0,C 180,E1 -20580.571,E2 -20580.571} C_VEL
LIN {X 0,Y 228.446,Z 249.018,A -85,B 0,C 180,E1 -20581.23,E2 -20581.23} C_VEL
LIN {X 0,Y 227.443,Z 254.372,A -85,B 0,C 180,E1 -20581.849,E2 -20581.849} C_VEL
LIN {X 0,Y 223.949,Z 266.388,A -85,B 0,C 180,E1 -20583.444,E2 -20583.444} C_VEL
LIN {X 0,Y 223.272,Z 271.176,A -85,B 0,C 180,E1 -20584.327,E2 -20584.327} C_VEL
LIN {X 0,Y 221.214,Z 279.944,A -85,B 0,C 180,E1 -20586.108,E2 -20586.108} C_VEL
LIN {X 0,Y 218.808,Z 289.192,A -85,B 0,C 180,E1 -20588.425,E2 -20588.425} C_VEL
LIN {X 0,Y 216.631,Z 297.577,A -85,B 0,C 180,E1 -20591.072,E2 -20591.072} C_VEL
LIN {X 0,Y 214.692,Z 304.522,A -85,B 0,C 180,E1 -20593.847,E2 -20593.847} C_VEL
LIN {X 0,Y 213.179,Z 310.089,A -85,B 0,C 180,E1 -20596.66,E2 -20596.66} C_VEL
LIN {X 0,Y 212.286,Z 314.465,A -85,B 0,C 180,E1 -20599.511,E2 -20599.511} C_VEL
LIN {X 0,Y 211.687,Z 317.763,A -85,B 0,C 180,E1 -20602.37,E2 -20602.37} C_VEL
LIN {X 0,Y 211.392,Z 320.446,A -85,B 0,C 180,E1 -20605.857,E2 -20605.857} C_VEL
LIN {X 0,Y 211.442,Z 321.461,A -85,B 0,C 180,E1 -20608.097,E2 -20608.097} C_VEL
LIN {X 0,Y 211.545,Z 321.855,A -85,B 0,C 180,E1 -20610.001,E2 -20610.001} C_VEL
LIN {X 0,Y 211.436,Z 321.854,A -85,B 0,C 180,E1 -20611.906,E2 -20611.906} C_VEL
LIN {X 0,Y 211.393,Z 321.371,A -85,B 0,C 180,E1 -20614.146,E2 -20614.146} C_VEL
LIN {X 0,Y 211.69,Z 319.459,A -85,B 0,C 180,E1 -20617.632,E2 -20617.632} C_VEL
LIN {X 0,Y 212.342,Z 316.872,A -85,B 0,C 180,E1 -20620.489,E2 -20620.489} C_VEL
LIN {X 0,Y 213.314,Z 313.277,A -85,B 0,C 180,E1 -20623.334,E2 -20623.334} C_VEL
LIN {X 0,Y 214.868,Z 308.585,A -85,B 0,C 180,E1 -20626.142,E2 -20626.142} C_VEL
LIN {X 0,Y 216.857,Z 302.651,A -85,B 0,C 180,E1 -20628.91,E2 -20628.91} C_VEL
LIN {X 0,Y 219.263,Z 295.239,A -85,B 0,C 180,E1 -20631.638,E2 -20631.638} C_VEL
LIN {X 0,Y 222.145,Z 286.099,A -85,B 0,C 180,E1 -20634.285,E2 -20634.285} C_VEL
LIN {X 0,Y 225.317,Z 275.51,A -85,B 0,C 180,E1 -20636.639,E2 -20636.639} C_VEL
LIN {X 0,Y 225.692,Z 270.994,A -85,B 0,C 180,E1 -20637.593,E2 -20637.593} C_VEL
LIN {X 0,Y 225.569,Z 260.788,A -85,B 0,C 180,E1 -20639.591,E2 -20639.591} C_VEL
LIN {X 0,Y 224.615,Z 250.172,A -85,B 0,C 180,E1 -20641.432,E2 -20641.432} C_VEL
LIN {X 0,Y 222.679,Z 238.715,A -85,B 0,C 180,E1 -20643.22,E2 -20643.22} C_VEL
LIN {X 0,Y 219.802,Z 227.242,A -85,B 0,C 180,E1 -20644.857,E2 -20644.857} C_VEL
LIN {X 0,Y 216.716,Z 218.432,A -85,B 0,C 180,E1 -20646.08,E2 -20646.08} C_VEL
LIN {X 0,Y 215.66,Z 215.021,A -85,B 0,C 180,E1 -20646.532,E2 -20646.532} C_VEL
LIN {X 0,Y 215.692,Z 213.258,A -85,B 0,C 180,E1 -20648.556,E2 -20648.556} C_VEL
LIN {X 0,Y 215.474,Z 210.913,A -85,B 0,C 180,E1 -20651.394,E2 -20651.394} C_VEL
LIN {X 0,Y 215.162,Z 208.846,A -85,B 0,C 180,E1 -20654.061,E2 -20654.061} C_VEL
LIN {X 0,Y 214.502,Z 205.202,A -85,B 0,C 180,E1 -20659.059,E2 -20659.059} C_VEL
LIN {X 0,Y 214.025,Z 202.076,A -85,B 0,C 180,E1 -20663.767,E2 -20663.767} C_VEL
LIN {X 0,Y 213.748,Z 200.864,A -85,B 0,C 180,E1 -20666.017,E2 -20666.017} C_VEL
LIN {X 0,Y 213.746,Z 200.863,A -85,B 0,C 180,E1 -20670.449,E2 -20670.449} C_VEL
LIN {X 0,Y 213.797,Z 200.855,A -85,B 0,C 180,E1 -20674.702,E2 -20674.702} C_VEL
LIN {X 0,Y 213.845,Z 200.848,A -85,B 0,C 180,E1 -20678.807,E2 -20678.807} C_VEL
LIN {X 0,Y 213.959,Z 200.834,A -85,B 0,C 180,E1 -20682.805,E2 -20682.805} C_VEL
LIN {X 0,Y 213.94,Z 200.837,A -85,B 0,C 180,E1 -20686.706,E2 -20686.706} C_VEL
LIN {X 0,Y 214.13,Z 200.812,A -85,B 0,C 180,E1 -20690.555,E2 -20690.555} C_VEL
LIN {X 0,Y 214.087,Z 200.818,A -85,B 0,C 180,E1 -20694.349,E2 -20694.349} C_VEL
LIN {X 0,Y 214.43,Z 200.774,A -85,B 0,C 180,E1 -20698.122,E2 -20698.122} C_VEL
LIN {X 0,Y 214.467,Z 200.77,A -85,B 0,C 180,E1 -20701.878,E2 -20701.878} C_VEL
LIN {X 0,Y 214.18,Z 200.805,A -85,B 0,C 180,E1 -20707.543,E2 -20707.543} C_VEL
LIN {X 0,Y 213.983,Z 200.831,A -85,B 0,C 180,E1 -20711.366,E2 -20711.366} C_VEL
LIN {X 0,Y 213.912,Z 200.837,A -85,B 0,C 180,E1 -20715.239,E2 -20715.239} C_VEL
LIN {X 0,Y 213.829,Z 200.85,A -85,B 0,C 180,E1 -20719.189,E2 -20719.189} C_VEL
LIN {X 0,Y 213.822,Z 200.851,A -85,B 0,C 180,E1 -20723.231,E2 -20723.231} C_VEL
LIN {X 0,Y 213.823,Z 200.852,A -85,B 0,C 180,E1 -20727.451,E2 -20727.451} C_VEL
LIN {X 0,Y 213.761,Z 200.858,A -85,B 0,C 180,E1 -20731.739,E2 -20731.739} C_VEL
LIN {X 0,Y 213.739,Z 200.862,A -85,B 0,C 180,E1 -20736.29,E2 -20736.29} C_VEL
LIN {X 0,Y 213.706,Z 200.865,A -85,B 0,C 180,E1 -20741.127,E2 -20741.127} C_VEL
LIN {X 0,Y 213.806,Z 201.553,A -85,B 0,C 180,E1 -20743.687,E2 -20743.687} C_VEL
LIN {X 0,Y 214.031,Z 203.101,A -85,B 0,C 180,E1 -20746.407,E2 -20746.407} C_VEL
LIN {X 0,Y 214.272,Z 205.437,A -85,B 0,C 180,E1 -20750.241,E2 -20750.241} C_VEL
LIN {X 0,Y 214.238,Z 206.097,A -85,B 0,C 180,E1 -20751.261,E2 -20751.261} C_VEL
LIN {X 0,Y 215.4,Z 209.345,A -85,B 0,C 180,E1 -20751.731,E2 -20751.731} C_VEL
LIN {X 0,Y 216.939,Z 212.495,A -85,B 0,C 180,E1 -20752.249,E2 -20752.249} C_VEL
LIN {X 0,Y 220.274,Z 220.803,A -85,B 0,C 180,E1 -20753.595,E2 -20753.595} C_VEL
LIN {X 0,Y 223.583,Z 231.194,A -85,B 0,C 180,E1 -20755.315,E2 -20755.315} C_VEL
LIN {X 0,Y 225.95,Z 241.524,A -85,B 0,C 180,E1 -20757.122,E2 -20757.122} C_VEL
LIN {X 0,Y 227.395,Z 251.795,A -85,B 0,C 180,E1 -20759.068,E2 -20759.068} C_VEL
LIN {X 0,Y 227.787,Z 259.579,A -85,B 0,C 180,E1 -20760.674,E2 -20760.674} C_VEL
LIN {X 0,Y 225.134,Z 269.216,A -85,B 0,C 180,E1 -20762.585,E2 -20762.585} C_VEL
LIN {X 0,Y 222.512,Z 277.985,A -85,B 0,C 180,E1 -20764.762,E2 -20764.762} C_VEL
LIN {X 0,Y 219.633,Z 286.512,A -85,B 0,C 180,E1 -20767.42,E2 -20767.42} C_VEL
LIN {X 0,Y 217.101,Z 293.829,A -85,B 0,C 180,E1 -20770.377,E2 -20770.377} C_VEL
LIN {X 0,Y 215.445,Z 298.765,A -85,B 0,C 180,E1 -20772.927,E2 -20772.927} C_VEL
LIN {X 0,Y 213.838,Z 303.024,A -85,B 0,C 180,E1 -20775.73,E2 -20775.73} C_VEL
LIN {X 0,Y 212.767,Z 306.217,A -85,B 0,C 180,E1 -20778.569,E2 -20778.569} C_VEL
LIN {X 0,Y 211.879,Z 308.986,A -85,B 0,C 180,E1 -20782.375,E2 -20782.375} C_VEL
LIN {X 0,Y 211.592,Z 309.954,A -85,B 0,C 180,E1 -20785.178,E2 -20785.178} C_VEL
LIN {X 0,Y 211.534,Z 310.065,A -85,B 0,C 180,E1 -20788.095,E2 -20788.095} C_VEL
LIN {X 0,Y 211.578,Z 309.665,A -85,B 0,C 180,E1 -20789.999,E2 -20789.999} C_VEL
LIN {X 0,Y 211.693,Z 308.844,A -85,B 0,C 180,E1 -20791.901,E2 -20791.901} C_VEL
LIN {X 0,Y 211.954,Z 307.616,A -85,B 0,C 180,E1 -20793.801,E2 -20793.801} C_VEL
LIN {X 0,Y 212.504,Z 305.022,A -85,B 0,C 180,E1 -20796.643,E2 -20796.643} C_VEL
LIN {X 0,Y 213.36,Z 301.426,A -85,B 0,C 180,E1 -20799.478,E2 -20799.478} C_VEL
LIN {X 0,Y 214.627,Z 296.727,A -85,B 0,C 180,E1 -20802.287,E2 -20802.287} C_VEL
LIN {X 0,Y 216.644,Z 289.673,A -85,B 0,C 180,E1 -20805.521,E2 -20805.521} C_VEL
LIN {X 0,Y 218.897,Z 281.99,A -85,B 0,C 180,E1 -20808.24,E2 -20808.24} C_VEL
LIN {X 0,Y 221.495,Z 272.362,A -85,B 0,C 180,E1 -20810.911,E2 -20810.911} C_VEL
LIN {X 0,Y 223.86,Z 262.418,A -85,B 0,C 180,E1 -20813.103,E2 -20813.103} C_VEL
LIN {X 0,Y 225.333,Z 255.988,A -85,B 0,C 180,E1 -20814.253,E2 -20814.253} C_VEL
LIN {X 0,Y 225.252,Z 250.952,A -85,B 0,C 180,E1 -20815.2,E2 -20815.2} C_VEL
LIN {X 0,Y 224.048,Z 241.36,A -85,B 0,C 180,E1 -20816.913,E2 -20816.913} C_VEL
LIN {X 0,Y 222.041,Z 231.127,A -85,B 0,C 180,E1 -20818.554,E2 -20818.554} C_VEL
LIN {X 0,Y 218.487,Z 218.323,A -85,B 0,C 180,E1 -20820.404,E2 -20820.404} C_VEL
LIN {X 0,Y 213.874,Z 206.208,A -85,B 0,C 180,E1 -20822.025,E2 -20822.025} C_VEL
LIN {X 0,Y 213.843,Z 205.821,A -85,B 0,C 180,E1 -20822.136,E2 -20822.136} C_VEL
LIN {X 0,Y 213.964,Z 203.982,A -85,B 0,C 180,E1 -20824.797,E2 -20824.797} C_VEL
LIN {X 0,Y 213.786,Z 201.518,A -85,B 0,C 180,E1 -20828.648,E2 -20828.648} C_VEL
LIN {X 0,Y 213.707,Z 200.865,A -85,B 0,C 180,E1 -20831.121,E2 -20831.121} C_VEL
LIN {X 0,Y 213.739,Z 200.863,A -85,B 0,C 180,E1 -20833.664,E2 -20833.664} C_VEL
LIN {X 0,Y 213.802,Z 200.853,A -85,B 0,C 180,E1 -20836.345,E2 -20836.345} C_VEL
LIN {X 0,Y 213.787,Z 200.858,A -85,B 0,C 180,E1 -20839.115,E2 -20839.115} C_VEL
LIN {X 0,Y 213.733,Z 200.861,A -85,B 0,C 180,E1 -20843.709,E2 -20843.709} C_VEL
LIN {X 0,Y 213.766,Z 200.857,A -85,B 0,C 180,E1 -20848.729,E2 -20848.729} C_VEL
LIN {X 0,Y 213.811,Z 200.852,A -85,B 0,C 180,E1 -20852.601,E2 -20852.601} C_VEL
LIN {X 0,Y 213.851,Z 200.824,A -85,B 0,C 180,E1 -20856.941,E2 -20856.941} C_VEL
LIN {X 0,Y 213.951,Z 200.822,A -85,B 0,C 180,E1 -20862.804,E2 -20862.804} C_VEL
LIN {X 0,Y 213.966,Z 200.83,A -85,B 0,C 180,E1 -20866.707,E2 -20866.707} C_VEL
LIN {X 0,Y 214.19,Z 200.799,A -85,B 0,C 180,E1 -20870.557,E2 -20870.557} C_VEL
LIN {X 0,Y 214.233,Z 200.799,A -85,B 0,C 180,E1 -20872.459,E2 -20872.459} C_VEL
LIN {X 0,Y 214.422,Z 200.771,A -85,B 0,C 180,E1 -20878.121,E2 -20878.121} C_VEL
LIN {X 0,Y 214.458,Z 200.772,A -85,B 0,C 180,E1 -20881.878,E2 -20881.878} C_VEL
LIN {X 0,Y 214.206,Z 200.804,A -85,B 0,C 180,E1 -20887.541,E2 -20887.541} C_VEL
LIN {X 0,Y 214.001,Z 200.83,A -85,B 0,C 180,E1 -20891.364,E2 -20891.364} C_VEL
LIN {X 0,Y 213.902,Z 200.843,A -85,B 0,C 180,E1 -20895.239,E2 -20895.239} C_VEL
LIN {X 0,Y 213.863,Z 200.847,A -85,B 0,C 180,E1 -20899.185,E2 -20899.185} C_VEL
LIN {X 0,Y 213.843,Z 200.849,A -85,B 0,C 180,E1 -20903.227,E2 -20903.227} C_VEL
LIN {X 0,Y 213.813,Z 200.851,A -85,B 0,C 180,E1 -20907.452,E2 -20907.452} C_VEL
LIN {X 0,Y 213.755,Z 200.847,A -85,B 0,C 180,E1 -20911.739,E2 -20911.739} C_VEL
LIN {X 0,Y 213.739,Z 200.862,A -85,B 0,C 180,E1 -20916.289,E2 -20916.289} C_VEL
LIN {X 0,Y 213.798,Z 200.991,A -85,B 0,C 180,E1 -20918.424,E2 -20918.424} C_VEL
LIN {X 0,Y 214.175,Z 202.803,A -85,B 0,C 180,E1 -20921.017,E2 -20921.017} C_VEL
LIN {X 0,Y 214.806,Z 206.573,A -85,B 0,C 180,E1 -20926.037,E2 -20926.037} C_VEL
LIN {X 0,Y 215.182,Z 209.134,A -85,B 0,C 180,E1 -20929.221,E2 -20929.221} C_VEL
LIN {X 0,Y 215.391,Z 212.269,A -85,B 0,C 180,E1 -20932.874,E2 -20932.874} C_VEL
LIN {X 0,Y 214.967,Z 215.248,A -85,B 0,C 180,E1 -20936.127,E2 -20936.127} C_VEL
LIN {X 0,Y 216.802,Z 221.712,A -85,B 0,C 180,E1 -20936.841,E2 -20936.841} C_VEL
LIN {X 0,Y 219.802,Z 233.115,A -85,B 0,C 180,E1 -20938.23,E2 -20938.23} C_VEL
LIN {X 0,Y 222.056,Z 245.984,A -85,B 0,C 180,E1 -20939.991,E2 -20939.991} C_VEL
LIN {X 0,Y 223.178,Z 257.832,A -85,B 0,C 180,E1 -20941.852,E2 -20941.852} C_VEL
LIN {X 0,Y 223.326,Z 268.915,A -85,B 0,C 180,E1 -20943.863,E2 -20943.863} C_VEL
LIN {X 0,Y 223.272,Z 271.176,A -85,B 0,C 180,E1 -20944.327,E2 -20944.327} C_VEL
LIN {X 0,Y 222.744,Z 274.285,A -85,B 0,C 180,E1 -20944.932,E2 -20944.932} C_VEL
LIN {X 0,Y 220.659,Z 278.781,A -85,B 0,C 180,E1 -20945.758,E2 -20945.758} C_VEL
LIN {X 0,Y 213.65,Z 288.416,A -85,B 0,C 180,E1 -20947.706,E2 -20947.706} C_VEL
LIN {X 0,Y 211.412,Z 292.308,A -85,B 0,C 180,E1 -20948.766,E2 -20948.766} C_VEL
LIN {X 0,Y 210.986,Z 293.566,A -85,B 0,C 180,E1 -20949.167,E2 -20949.167} C_VEL
LIN {X 0,Y 208.839,Z 300.967,A -85,B 0,C 180,E1 -20951.866,E2 -20951.866} C_VEL
LIN {X 0,Y 206.707,Z 308.118,A -85,B 0,C 180,E1 -20955.229,E2 -20955.229} C_VEL
LIN {X 0,Y 205.541,Z 312.892,A -85,B 0,C 180,E1 -20958.164,E2 -20958.164} C_VEL
LIN {X 0,Y 204.81,Z 316.546,A -85,B 0,C 180,E1 -20961.119,E2 -20961.119} C_VEL
LIN {X 0,Y 204.401,Z 319.184,A -85,B 0,C 180,E1 -20964.081,E2 -20964.081} C_VEL
LIN {X 0,Y 204.295,Z 320.428,A -85,B 0,C 180,E1 -20966.056,E2 -20966.056} C_VEL
LIN {X 0,Y 204.344,Z 321.255,A -85,B 0,C 180,E1 -20968.031,E2 -20968.031} C_VEL
LIN {X 0,Y 204.462,Z 321.655,A -85,B 0,C 180,E1 -20970.001,E2 -20970.001} C_VEL
LIN {X 0,Y 204.339,Z 321.659,A -85,B 0,C 180,E1 -20971.972,E2 -20971.972} C_VEL
LIN {X 0,Y 204.296,Z 321.279,A -85,B 0,C 180,E1 -20973.946,E2 -20973.946} C_VEL
LIN {X 0,Y 204.402,Z 320.501,A -85,B 0,C 180,E1 -20975.921,E2 -20975.921} C_VEL
LIN {X 0,Y 205.068,Z 317.665,A -85,B 0,C 180,E1 -20979.867,E2 -20979.867} C_VEL
LIN {X 0,Y 205.99,Z 314.421,A -85,B 0,C 180,E1 -20982.813,E2 -20982.813} C_VEL
LIN {X 0,Y 207.397,Z 310.118,A -85,B 0,C 180,E1 -20985.73,E2 -20985.73} C_VEL
LIN {X 0,Y 209.437,Z 304.641,A -85,B 0,C 180,E1 -20988.59,E2 -20988.59} C_VEL
LIN {X 0,Y 212.062,Z 297.037,A -85,B 0,C 180,E1 -20991.691,E2 -20991.691} C_VEL
LIN {X 0,Y 214.599,Z 289.284,A -85,B 0,C 180,E1 -20994.165,E2 -20994.165} C_VEL
LIN {X 0,Y 217.422,Z 280.537,A -85,B 0,C 180,E1 -20996.388,E2 -20996.388} C_VEL
LIN {X 0,Y 218.977,Z 275.45,A -85,B 0,C 180,E1 -20997.474,E2 -20997.474} C_VEL
LIN {X 0,Y 219.209,Z 266.425,A -85,B 0,C 180,E1 -20999.443,E2 -20999.443} C_VEL
LIN {X 0,Y 218.72,Z 255.829,A -85,B 0,C 180,E1 -21001.485,E2 -21001.485} C_VEL
LIN {X 0,Y 217.206,Z 243.999,A -85,B 0,C 180,E1 -21003.522,E2 -21003.522} C_VEL
LIN {X 0,Y 214.96,Z 233.486,A -85,B 0,C 180,E1 -21005.179,E2 -21005.179} C_VEL
LIN {X 0,Y 211.707,Z 222.66,A -85,B 0,C 180,E1 -21006.804,E2 -21006.804} C_VEL
LIN {X 0,Y 209.746,Z 218.115,A -85,B 0,C 180,E1 -21007.534,E2 -21007.534} C_VEL
LIN {X 0,Y 208.655,Z 214.78,A -85,B 0,C 180,E1 -21008.011,E2 -21008.011} C_VEL
LIN {X 0,Y 208.339,Z 211.308,A -85,B 0,C 180,E1 -21012.426,E2 -21012.426} C_VEL
LIN {X 0,Y 207.982,Z 209.246,A -85,B 0,C 180,E1 -21015.202,E2 -21015.202} C_VEL
LIN {X 0,Y 207.395,Z 205.939,A -85,B 0,C 180,E1 -21019.921,E2 -21019.921} C_VEL
LIN {X 0,Y 207.194,Z 204.371,A -85,B 0,C 180,E1 -21022.37,E2 -21022.37} C_VEL
LIN {X 0,Y 206.687,Z 201.745,A -85,B 0,C 180,E1 -21027.041,E2 -21027.041} C_VEL
LIN {X 0,Y 206.745,Z 201.733,A -85,B 0,C 180,E1 -21032.103,E2 -21032.103} C_VEL
LIN {X 0,Y 206.788,Z 201.728,A -85,B 0,C 180,E1 -21036.576,E2 -21036.576} C_VEL
LIN {X 0,Y 206.875,Z 201.717,A -85,B 0,C 180,E1 -21042.197,E2 -21042.197} C_VEL
LIN {X 0,Y 206.883,Z 201.715,A -85,B 0,C 180,E1 -21046.244,E2 -21046.244} C_VEL
LIN {X 0,Y 207.09,Z 201.688,A -85,B 0,C 180,E1 -21050.231,E2 -21050.231} C_VEL
LIN {X 0,Y 207.048,Z 201.696,A -85,B 0,C 180,E1 -21054.156,E2 -21054.156} C_VEL
LIN {X 0,Y 207.367,Z 201.653,A -85,B 0,C 180,E1 -21058.058,E2 -21058.058} C_VEL
LIN {X 0,Y 207.491,Z 201.639,A -85,B 0,C 180,E1 -21060,E2 -21060} C_VEL
LIN {X 0,Y 207.4,Z 201.651,A -85,B 0,C 180,E1 -21061.942,E2 -21061.942} C_VEL
LIN {X 0,Y 207.122,Z 201.686,A -85,B 0,C 180,E1 -21067.801,E2 -21067.801} C_VEL
LIN {X 0,Y 206.907,Z 201.711,A -85,B 0,C 180,E1 -21071.76,E2 -21071.76} C_VEL
LIN {X 0,Y 206.849,Z 201.72,A -85,B 0,C 180,E1 -21075.773,E2 -21075.773} C_VEL
LIN {X 0,Y 206.774,Z 201.728,A -85,B 0,C 180,E1 -21079.871,E2 -21079.871} C_VEL
LIN {X 0,Y 206.748,Z 201.73,A -85,B 0,C 180,E1 -21084.075,E2 -21084.075} C_VEL
LIN {X 0,Y 206.731,Z 201.732,A -85,B 0,C 180,E1 -21088.421,E2 -21088.421} C_VEL
LIN {X 0,Y 206.693,Z 201.74,A -85,B 0,C 180,E1 -21092.959,E2 -21092.959} C_VEL
LIN {X 0,Y 206.674,Z 201.738,A -85,B 0,C 180,E1 -21097.742,E2 -21097.742} C_VEL
LIN {X 0,Y 206.659,Z 201.754,A -85,B 0,C 180,E1 -21101.571,E2 -21101.571} C_VEL
LIN {X 0,Y 206.937,Z 203.87,A -85,B 0,C 180,E1 -21105.497,E2 -21105.497} C_VEL
LIN {X 0,Y 207.301,Z 206.519,A -85,B 0,C 180,E1 -21109.803,E2 -21109.803} C_VEL
LIN {X 0,Y 208.454,Z 209.595,A -85,B 0,C 180,E1 -21110.266,E2 -21110.266} C_VEL
LIN {X 0,Y 209.629,Z 211.783,A -85,B 0,C 180,E1 -21110.674,E2 -21110.674} C_VEL
LIN {X 0,Y 213.648,Z 221.106,A -85,B 0,C 180,E1 -21112.331,E2 -21112.331} C_VEL
LIN {X 0,Y 217.361,Z 232.946,A -85,B 0,C 180,E1 -21114.41,E2 -21114.41} C_VEL
LIN {X 0,Y 219.619,Z 243.135,A -85,B 0,C 180,E1 -21116.309,E2 -21116.309} C_VEL
LIN {X 0,Y 220.983,Z 253.29,A -85,B 0,C 180,E1 -21118.35,E2 -21118.35} C_VEL
LIN {X 0,Y 221.29,Z 260.778,A -85,B 0,C 180,E1 -21119.987,E2 -21119.987} C_VEL
LIN {X 0,Y 218.278,Z 271.209,A -85,B 0,C 180,E1 -21122.17,E2 -21122.17} C_VEL
LIN {X 0,Y 215.573,Z 279.634,A -85,B 0,C 180,E1 -21124.408,E2 -21124.408} C_VEL
LIN {X 0,Y 212.626,Z 287.847,A -85,B 0,C 180,E1 -21127.147,E2 -21127.147} C_VEL
LIN {X 0,Y 210.326,Z 294.142,A -85,B 0,C 180,E1 -21129.814,E2 -21129.814} C_VEL
LIN {X 0,Y 208.643,Z 298.904,A -85,B 0,C 180,E1 -21132.353,E2 -21132.353} C_VEL
LIN {X 0,Y 206.92,Z 303.177,A -85,B 0,C 180,E1 -21135.242,E2 -21135.242} C_VEL
LIN {X 0,Y 205.797,Z 306.383,A -85,B 0,C 180,E1 -21138.176,E2 -21138.176} C_VEL
LIN {X 0,Y 204.843,Z 309.165,A -85,B 0,C 180,E1 -21142.111,E2 -21142.111} C_VEL
LIN {X 0,Y 204.504,Z 310.209,A -85,B 0,C 180,E1 -21145.294,E2 -21145.294} C_VEL
LIN {X 0,Y 204.436,Z 310.266,A -85,B 0,C 180,E1 -21148.029,E2 -21148.029} C_VEL
LIN {X 0,Y 204.496,Z 309.871,A -85,B 0,C 180,E1 -21149.999,E2 -21149.999} C_VEL
LIN {X 0,Y 204.617,Z 309.062,A -85,B 0,C 180,E1 -21151.967,E2 -21151.967} C_VEL
LIN {X 0,Y 204.89,Z 307.84,A -85,B 0,C 180,E1 -21153.932,E2 -21153.932} C_VEL
LIN {X 0,Y 205.364,Z 305.675,A -85,B 0,C 180,E1 -21156.485,E2 -21156.485} C_VEL
LIN {X 0,Y 206.385,Z 301.675,A -85,B 0,C 180,E1 -21159.801,E2 -21159.801} C_VEL
LIN {X 0,Y 207.716,Z 296.99,A -85,B 0,C 180,E1 -21162.702,E2 -21162.702} C_VEL
LIN {X 0,Y 209.838,Z 289.952,A -85,B 0,C 180,E1 -21166.038,E2 -21166.038} C_VEL
LIN {X 0,Y 212.178,Z 282.296,A -85,B 0,C 180,E1 -21168.839,E2 -21168.839} C_VEL
LIN {X 0,Y 214.901,Z 272.689,A -85,B 0,C 180,E1 -21171.584,E2 -21171.584} C_VEL
LIN {X 0,Y 217.372,Z 262.776,A -85,B 0,C 180,E1 -21173.834,E2 -21173.834} C_VEL
LIN {X 0,Y 218.819,Z 256.733,A -85,B 0,C 180,E1 -21174.953,E2 -21174.953} C_VEL
LIN {X 0,Y 218.313,Z 248.558,A -85,B 0,C 180,E1 -21176.579,E2 -21176.579} C_VEL
LIN {X 0,Y 216.808,Z 238.17,A -85,B 0,C 180,E1 -21178.444,E2 -21178.444} C_VEL
LIN {X 0,Y 214.273,Z 227.299,A -85,B 0,C 180,E1 -21180.223,E2 -21180.223} C_VEL
LIN {X 0,Y 211.358,Z 217.652,A -85,B 0,C 180,E1 -21181.676,E2 -21181.676} C_VEL
LIN {X 0,Y 207.819,Z 209.004,A -85,B 0,C 180,E1 -21182.956,E2 -21182.956} C_VEL
LIN {X 0,Y 206.875,Z 206.066,A -85,B 0,C 180,E1 -21183.346,E2 -21183.346} C_VEL
LIN {X 0,Y 206.922,Z 204.731,A -85,B 0,C 180,E1 -21185.397,E2 -21185.397} C_VEL
LIN {X 0,Y 206.813,Z 202.749,A -85,B 0,C 180,E1 -21188.592,E2 -21188.592} C_VEL
LIN {X 0,Y 206.638,Z 201.777,A -85,B 0,C 180,E1 -21190.251,E2 -21190.251} C_VEL
LIN {X 0,Y 206.7,Z 201.736,A -85,B 0,C 180,E1 -21195.557,E2 -21195.557} C_VEL
LIN {X 0,Y 206.716,Z 201.735,A -85,B 0,C 180,E1 -21199.761,E2 -21199.761} C_VEL
LIN {X 0,Y 206.713,Z 201.735,A -85,B 0,C 180,E1 -21202.266,E2 -21202.266} C_VEL
LIN {X 0,Y 206.686,Z 201.738,A -85,B 0,C 180,E1 -21207.039,E2 -21207.039} C_VEL
LIN {X 0,Y 206.75,Z 201.729,A -85,B 0,C 180,E1 -21212.095,E2 -21212.095} C_VEL
LIN {X 0,Y 206.781,Z 201.706,A -85,B 0,C 180,E1 -21216.574,E2 -21216.574} C_VEL
LIN {X 0,Y 206.87,Z 201.697,A -85,B 0,C 180,E1 -21222.018,E2 -21222.018} C_VEL
LIN {X 0,Y 206.899,Z 201.713,A -85,B 0,C 180,E1 -21226.244,E2 -21226.244} C_VEL
LIN {X 0,Y 207.125,Z 201.675,A -85,B 0,C 180,E1 -21230.232,E2 -21230.232} C_VEL
LIN {X 0,Y 207.175,Z 201.68,A -85,B 0,C 180,E1 -21232.201,E2 -21232.201} C_VEL
LIN {X 0,Y 207.359,Z 201.65,A -85,B 0,C 180,E1 -21238.057,E2 -21238.057} C_VEL
LIN {X 0,Y 207.485,Z 201.641,A -85,B 0,C 180,E1 -21240,E2 -21240} C_VEL
LIN {X 0,Y 207.391,Z 201.652,A -85,B 0,C 180,E1 -21241.942,E2 -21241.942} C_VEL
LIN {X 0,Y 207.146,Z 201.684,A -85,B 0,C 180,E1 -21247.799,E2 -21247.799} C_VEL
LIN {X 0,Y 206.92,Z 201.711,A -85,B 0,C 180,E1 -21251.758,E2 -21251.758} C_VEL
LIN {X 0,Y 206.838,Z 201.722,A -85,B 0,C 180,E1 -21255.773,E2 -21255.773} C_VEL
LIN {X 0,Y 206.802,Z 201.726,A -85,B 0,C 180,E1 -21259.867,E2 -21259.867} C_VEL
LIN {X 0,Y 206.754,Z 201.731,A -85,B 0,C 180,E1 -21264.073,E2 -21264.073} C_VEL
LIN {X 0,Y 206.728,Z 201.731,A -85,B 0,C 180,E1 -21268.421,E2 -21268.421} C_VEL
LIN {X 0,Y 206.69,Z 201.738,A -85,B 0,C 180,E1 -21272.959,E2 -21272.959} C_VEL
LIN {X 0,Y 206.743,Z 201.904,A -85,B 0,C 180,E1 -21277.726,E2 -21277.726} C_VEL
LIN {X 0,Y 207.256,Z 204.623,A -85,B 0,C 180,E1 -21281.76,E2 -21281.76} C_VEL
LIN {X 0,Y 207.688,Z 207.192,A -85,B 0,C 180,E1 -21285.285,E2 -21285.285} C_VEL
LIN {X 0,Y 207.999,Z 209.286,A -85,B 0,C 180,E1 -21288.017,E2 -21288.017} C_VEL
LIN {X 0,Y 208.282,Z 211.6,A -85,B 0,C 180,E1 -21290.903,E2 -21290.903} C_VEL
LIN {X 0,Y 208.291,Z 214.305,A -85,B 0,C 180,E1 -21294.075,E2 -21294.075} C_VEL
LIN {X 0,Y 208.145,Z 215.056,A -85,B 0,C 180,E1 -21294.917,E2 -21294.917} C_VEL
LIN {X 0,Y 209.166,Z 218.58,A -85,B 0,C 180,E1 -21295.331,E2 -21295.331} C_VEL
LIN {X 0,Y 212.636,Z 230.869,A -85,B 0,C 180,E1 -21296.885,E2 -21296.885} C_VEL
LIN {X 0,Y 215.026,Z 243.06,A -85,B 0,C 180,E1 -21298.59,E2 -21298.59} C_VEL
LIN {X 0,Y 216.307,Z 253.786,A -85,B 0,C 180,E1 -21300.284,E2 -21300.284} C_VEL
LIN {X 0,Y 216.712,Z 264.792,A -85,B 0,C 180,E1 -21302.256,E2 -21302.256} C_VEL
LIN {X 0,Y 216.414,Z 273.329,A -85,B 0,C 180,E1 -21304.001,E2 -21304.001} C_VEL
LIN {X 0,Y 213.672,Z 283.414,A -85,B 0,C 180,E1 -21306.242,E2 -21306.242} C_VEL
LIN {X 0,Y 211.182,Z 292.815,A -85,B 0,C 180,E1 -21308.918,E2 -21308.918} C_VEL
LIN {X 0,Y 210.986,Z 293.566,A -85,B 0,C 180,E1 -21309.167,E2 -21309.167} C_VEL
LIN {X 0,Y 209.357,Z 297.219,A -85,B 0,C 180,E1 -21310.366,E2 -21310.366} C_VEL
LIN {X 0,Y 204.909,Z 302.594,A -85,B 0,C 180,E1 -21312.317,E2 -21312.317} C_VEL
LIN {X 0,Y 200.592,Z 307.364,A -85,B 0,C 180,E1 -21314.46,E2 -21314.46} C_VEL
LIN {X 0,Y 199.211,Z 309.94,A -85,B 0,C 180,E1 -21315.933,E2 -21315.933} C_VEL
LIN {X 0,Y 198.248,Z 313.987,A -85,B 0,C 180,E1 -21318.759,E2 -21318.759} C_VEL
LIN {X 0,Y 197.588,Z 317.309,A -85,B 0,C 180,E1 -21321.822,E2 -21321.822} C_VEL
LIN {X 0,Y 197.34,Z 318.962,A -85,B 0,C 180,E1 -21323.869,E2 -21323.869} C_VEL
LIN {X 0,Y 197.19,Z 320.417,A -85,B 0,C 180,E1 -21326.32,E2 -21326.32} C_VEL
LIN {X 0,Y 197.362,Z 321.454,A -85,B 0,C 180,E1 -21330.001,E2 -21330.001} C_VEL
LIN {X 0,Y 197.203,Z 321.173,A -85,B 0,C 180,E1 -21333.738,E2 -21333.738} C_VEL
LIN {X 0,Y 197.341,Z 320.319,A -85,B 0,C 180,E1 -21336.134,E2 -21336.134} C_VEL
LIN {X 0,Y 198.04,Z 317.495,A -85,B 0,C 180,E1 -21340.221,E2 -21340.221} C_VEL
LIN {X 0,Y 199.043,Z 314.262,A -85,B 0,C 180,E1 -21343.269,E2 -21343.269} C_VEL
LIN {X 0,Y 200.56,Z 309.972,A -85,B 0,C 180,E1 -21346.28,E2 -21346.28} C_VEL
LIN {X 0,Y 202.673,Z 304.507,A -85,B 0,C 180,E1 -21349.234,E2 -21349.234} C_VEL
LIN {X 0,Y 205.18,Z 297.683,A -85,B 0,C 180,E1 -21352.134,E2 -21352.134} C_VEL
LIN {X 0,Y 208.113,Z 289.19,A -85,B 0,C 180,E1 -21354.968,E2 -21354.968} C_VEL
LIN {X 0,Y 211.087,Z 280.465,A -85,B 0,C 180,E1 -21357.244,E2 -21357.244} C_VEL
LIN {X 0,Y 212.483,Z 275.387,A -85,B 0,C 180,E1 -21358.389,E2 -21358.389} C_VEL
LIN {X 0,Y 212.719,Z 264.701,A -85,B 0,C 180,E1 -21360.795,E2 -21360.795} C_VEL
LIN {X 0,Y 212.081,Z 253.589,A -85,B 0,C 180,E1 -21362.986,E2 -21362.986} C_VEL
LIN {X 0,Y 210.387,Z 241.768,A -85,B 0,C 180,E1 -21365.071,E2 -21365.071} C_VEL
LIN {X 0,Y 207.495,Z 229.76,A -85,B 0,C 180,E1 -21367.055,E2 -21367.055} C_VEL
LIN {X 0,Y 204.738,Z 222.201,A -85,B 0,C 180,E1 -21368.346,E2 -21368.346} C_VEL
LIN {X 0,Y 203.161,Z 218.587,A -85,B 0,C 180,E1 -21368.974,E2 -21368.974} C_VEL
LIN {X 0,Y 201.735,Z 215.44,A -85,B 0,C 180,E1 -21369.53,E2 -21369.53} C_VEL
LIN {X 0,Y 201.565,Z 214.542,A -85,B 0,C 180,E1 -21369.69,E2 -21369.69} C_VEL
LIN {X 0,Y 201.072,Z 211.08,A -85,B 0,C 180,E1 -21374.349,E2 -21374.349} C_VEL
LIN {X 0,Y 200.63,Z 208.357,A -85,B 0,C 180,E1 -21378.275,E2 -21378.275} C_VEL
LIN {X 0,Y 200.061,Z 204.89,A -85,B 0,C 180,E1 -21383.895,E2 -21383.895} C_VEL
LIN {X 0,Y 199.678,Z 202.618,A -85,B 0,C 180,E1 -21388.133,E2 -21388.133} C_VEL
LIN {X 0,Y 199.672,Z 202.615,A -85,B 0,C 180,E1 -21392.77,E2 -21392.77} C_VEL
LIN {X 0,Y 199.748,Z 202.603,A -85,B 0,C 180,E1 -21397.231,E2 -21397.231} C_VEL
LIN {X 0,Y 199.83,Z 202.594,A -85,B 0,C 180,E1 -21401.721,E2 -21401.721} C_VEL
LIN {X 0,Y 199.826,Z 202.593,A -85,B 0,C 180,E1 -21405.748,E2 -21405.748} C_VEL
LIN {X 0,Y 200.014,Z 202.57,A -85,B 0,C 180,E1 -21409.882,E2 -21409.882} C_VEL
LIN {X 0,Y 200.01,Z 202.571,A -85,B 0,C 180,E1 -21413.949,E2 -21413.949} C_VEL
LIN {X 0,Y 200.307,Z 202.532,A -85,B 0,C 180,E1 -21417.99,E2 -21417.99} C_VEL
LIN {X 0,Y 200.457,Z 202.515,A -85,B 0,C 180,E1 -21420,E2 -21420} C_VEL
LIN {X 0,Y 200.336,Z 202.531,A -85,B 0,C 180,E1 -21422.011,E2 -21422.011} C_VEL
LIN {X 0,Y 200.068,Z 202.564,A -85,B 0,C 180,E1 -21428.078,E2 -21428.078} C_VEL
LIN {X 0,Y 199.858,Z 202.588,A -85,B 0,C 180,E1 -21432.181,E2 -21432.181} C_VEL
LIN {X 0,Y 199.789,Z 202.598,A -85,B 0,C 180,E1 -21436.345,E2 -21436.345} C_VEL
LIN {X 0,Y 199.691,Z 202.61,A -85,B 0,C 180,E1 -21440.607,E2 -21440.607} C_VEL
LIN {X 0,Y 199.662,Z 202.614,A -85,B 0,C 180,E1 -21444.986,E2 -21444.986} C_VEL
LIN {X 0,Y 199.658,Z 202.616,A -85,B 0,C 180,E1 -21449.526,E2 -21449.526} C_VEL
LIN {X 0,Y 199.666,Z 202.613,A -85,B 0,C 180,E1 -21452.356,E2 -21452.356} C_VEL
LIN {X 0,Y 199.618,Z 202.618,A -85,B 0,C 180,E1 -21456.765,E2 -21456.765} C_VEL
LIN {X 0,Y 199.603,Z 202.62,A -85,B 0,C 180,E1 -21459.33,E2 -21459.33} C_VEL
LIN {X 0,Y 199.717,Z 203.506,A -85,B 0,C 180,E1 -21462.357,E2 -21462.357} C_VEL
LIN {X 0,Y 199.96,Z 205.057,A -85,B 0,C 180,E1 -21465.339,E2 -21465.339} C_VEL
LIN {X 0,Y 200.171,Z 206.659,A -85,B 0,C 180,E1 -21468.113,E2 -21468.113} C_VEL
LIN {X 0,Y 201.468,Z 209.872,A -85,B 0,C 180,E1 -21468.658,E2 -21468.658} C_VEL
LIN {X 0,Y 202.76,Z 212.026,A -85,B 0,C 180,E1 -21469.124,E2 -21469.124} C_VEL
LIN {X 0,Y 207.467,Z 222.617,A -85,B 0,C 180,E1 -21471.182,E2 -21471.182} C_VEL
LIN {X 0,Y 210.762,Z 233.13,A -85,B 0,C 180,E1 -21473.16,E2 -21473.16} C_VEL
LIN {X 0,Y 213.063,Z 243.302,A -85,B 0,C 180,E1 -21475.163,E2 -21475.163} C_VEL
LIN {X 0,Y 214.493,Z 253.648,A -85,B 0,C 180,E1 -21477.349,E2 -21477.349} C_VEL
LIN {X 0,Y 214.806,Z 262.047,A -85,B 0,C 180,E1 -21479.272,E2 -21479.272} C_VEL
LIN {X 0,Y 212.013,Z 271.269,A -85,B 0,C 180,E1 -21481.272,E2 -21481.272} C_VEL
LIN {X 0,Y 209.174,Z 279.723,A -85,B 0,C 180,E1 -21483.565,E2 -21483.565} C_VEL
LIN {X 0,Y 206.056,Z 287.955,A -85,B 0,C 180,E1 -21486.375,E2 -21486.375} C_VEL
LIN {X 0,Y 203.572,Z 294.467,A -85,B 0,C 180,E1 -21489.219,E2 -21489.219} C_VEL
LIN {X 0,Y 201.865,Z 299.043,A -85,B 0,C 180,E1 -21491.739,E2 -21491.739} C_VEL
LIN {X 0,Y 200.032,Z 303.33,A -85,B 0,C 180,E1 -21494.721,E2 -21494.721} C_VEL
LIN {X 0,Y 198.843,Z 306.548,A -85,B 0,C 180,E1 -21497.756,E2 -21497.756} C_VEL
LIN {X 0,Y 197.784,Z 309.344,A -85,B 0,C 180,E1 -21501.828,E2 -21501.828} C_VEL
LIN {X 0,Y 197.407,Z 310.443,A -85,B 0,C 180,E1 -21505.456,E2 -21505.456} C_VEL
LIN {X 0,Y 197.34,Z 310.467,A -85,B 0,C 180,E1 -21507.958,E2 -21507.958} C_VEL
LIN {X 0,Y 197.397,Z 310.078,A -85,B 0,C 180,E1 -21509.999,E2 -21509.999} C_VEL
LIN {X 0,Y 197.542,Z 309.279,A -85,B 0,C 180,E1 -21512.037,E2 -21512.037} C_VEL
LIN {X 0,Y 197.809,Z 308.064,A -85,B 0,C 180,E1 -21514.073,E2 -21514.073} C_VEL
LIN {X 0,Y 198.578,Z 304.888,A -85,B 0,C 180,E1 -21517.7,E2 -21517.7} C_VEL
LIN {X 0,Y 199.816,Z 300.512,A -85,B 0,C 180,E1 -21521.152,E2 -21521.152} C_VEL
LIN {X 0,Y 201.336,Z 295.455,A -85,B 0,C 180,E1 -21524.141,E2 -21524.141} C_VEL
LIN {X 0,Y 203.428,Z 289.077,A -85,B 0,C 180,E1 -21527.074,E2 -21527.074} C_VEL
LIN {X 0,Y 205.944,Z 281.125,A -85,B 0,C 180,E1 -21529.951,E2 -21529.951} C_VEL
LIN {X 0,Y 208.341,Z 273.017,A -85,B 0,C 180,E1 -21532.299,E2 -21532.299} C_VEL
LIN {X 0,Y 210.898,Z 263.133,A -85,B 0,C 180,E1 -21534.614,E2 -21534.614} C_VEL
LIN {X 0,Y 212.077,Z 258.497,A -85,B 0,C 180,E1 -21535.515,E2 -21535.515} C_VEL
LIN {X 0,Y 212.209,Z 254.531,A -85,B 0,C 180,E1 -21536.328,E2 -21536.328} C_VEL
LIN {X 0,Y 211.121,Z 244.015,A -85,B 0,C 180,E1 -21538.436,E2 -21538.436} C_VEL
LIN {X 0,Y 208.981,Z 232.927,A -85,B 0,C 180,E1 -21540.435,E2 -21540.435} C_VEL
LIN {X 0,Y 205.912,Z 221.717,A -85,B 0,C 180,E1 -21542.281,E2 -21542.281} C_VEL
LIN {X 0,Y 201.472,Z 210.176,A -85,B 0,C 180,E1 -21544.117,E2 -21544.117} C_VEL
LIN {X 0,Y 200.103,Z 207.226,A -85,B 0,C 180,E1 -21544.597,E2 -21544.597} C_VEL
LIN {X 0,Y 199.925,Z 206.296,A -85,B 0,C 180,E1 -21544.729,E2 -21544.729} C_VEL
LIN {X 0,Y 199.723,Z 203.549,A -85,B 0,C 180,E1 -21549.296,E2 -21549.296} C_VEL
LIN {X 0,Y 199.585,Z 202.625,A -85,B 0,C 180,E1 -21552.312,E2 -21552.312} C_VEL
LIN {X 0,Y 199.637,Z 202.616,A -85,B 0,C 180,E1 -21555.244,E2 -21555.244} C_VEL
LIN {X 0,Y 199.658,Z 202.615,A -85,B 0,C 180,E1 -21558.024,E2 -21558.024} C_VEL
LIN {X 0,Y 199.67,Z 202.614,A -85,B 0,C 180,E1 -21560.74,E2 -21560.74} C_VEL
LIN {X 0,Y 199.6,Z 202.622,A -85,B 0,C 180,E1 -21565.71,E2 -21565.71} C_VEL
LIN {X 0,Y 199.679,Z 202.609,A -85,B 0,C 180,E1 -21568.132,E2 -21568.132} C_VEL
LIN {X 0,Y 199.673,Z 202.615,A -85,B 0,C 180,E1 -21572.769,E2 -21572.769} C_VEL
LIN {X 0,Y 199.739,Z 202.572,A -85,B 0,C 180,E1 -21577.229,E2 -21577.229} C_VEL
LIN {X 0,Y 199.822,Z 202.569,A -85,B 0,C 180,E1 -21581.72,E2 -21581.72} C_VEL
LIN {X 0,Y 199.834,Z 202.593,A -85,B 0,C 180,E1 -21585.748,E2 -21585.748} C_VEL
LIN {X 0,Y 200.066,Z 202.552,A -85,B 0,C 180,E1 -21589.883,E2 -21589.883} C_VEL
LIN {X 0,Y 200.119,Z 202.556,A -85,B 0,C 180,E1 -21591.924,E2 -21591.924} C_VEL
LIN {X 0,Y 200.299,Z 202.528,A -85,B 0,C 180,E1 -21597.989,E2 -21597.989} C_VEL
LIN {X 0,Y 200.45,Z 202.517,A -85,B 0,C 180,E1 -21600,E2 -21600} C_VEL
LIN {X 0,Y 200.328,Z 202.532,A -85,B 0,C 180,E1 -21602.01,E2 -21602.01} C_VEL
LIN {X 0,Y 200.09,Z 202.562,A -85,B 0,C 180,E1 -21608.076,E2 -21608.076} C_VEL
LIN {X 0,Y 200.018,Z 202.571,A -85,B 0,C 180,E1 -21610.348,E2 -21610.348} C_VEL
LIN {X 0,Y 199.78,Z 202.6,A -85,B 0,C 180,E1 -21616.345,E2 -21616.345} C_VEL
LIN {X 0,Y 199.809,Z 202.597,A -85,B 0,C 180,E1 -21618.455,E2 -21618.455} C_VEL
LIN {X 0,Y 199.729,Z 202.606,A -85,B 0,C 180,E1 -21623.824,E2 -21623.824} C_VEL
LIN {X 0,Y 199.697,Z 202.607,A -85,B 0,C 180,E1 -21628.388,E2 -21628.388} C_VEL
LIN {X 0,Y 199.642,Z 202.61,A -85,B 0,C 180,E1 -21632.351,E2 -21632.351} C_VEL
LIN {X 0,Y 199.69,Z 202.67,A -85,B 0,C 180,E1 -21636.748,E2 -21636.748} C_VEL
LIN {X 0,Y 200.291,Z 205.935,A -85,B 0,C 180,E1 -21641.812,E2 -21641.812} C_VEL
LIN {X 0,Y 200.699,Z 208.576,A -85,B 0,C 180,E1 -21645.551,E2 -21645.551} C_VEL
LIN {X 0,Y 201.22,Z 212.078,A -85,B 0,C 180,E1 -21650.209,E2 -21650.209} C_VEL
LIN {X 0,Y 201.275,Z 214.835,A -85,B 0,C 180,E1 -21653.592,E2 -21653.592} C_VEL
LIN {X 0,Y 202.249,Z 218.13,A -85,B 0,C 180,E1 -21653.997,E2 -21653.997} C_VEL
LIN {X 0,Y 205.54,Z 228.632,A -85,B 0,C 180,E1 -21655.439,E2 -21655.439} C_VEL
LIN {X 0,Y 208.23,Z 241.53,A -85,B 0,C 180,E1 -21657.319,E2 -21657.319} C_VEL
LIN {X 0,Y 209.646,Z 252.682,A -85,B 0,C 180,E1 -21659.139,E2 -21659.139} C_VEL
LIN {X 0,Y 210.125,Z 262.96,A -85,B 0,C 180,E1 -21661.025,E2 -21661.025} C_VEL
LIN {X 0,Y 209.899,Z 272.976,A -85,B 0,C 180,E1 -21663.13,E2 -21663.13} C_VEL
LIN {X 0,Y 207.157,Z 283.1,A -85,B 0,C 180,E1 -21665.447,E2 -21665.447} C_VEL
LIN {X 0,Y 204.674,Z 291.886,A -85,B 0,C 180,E1 -21667.989,E2 -21667.989} C_VEL
LIN {X 0,Y 202.795,Z 298.261,A -85,B 0,C 180,E1 -21670.254,E2 -21670.254} C_VEL
LIN {X 0,Y 200.717,Z 305.009,A -85,B 0,C 180,E1 -21673.212,E2 -21673.212} C_VEL
LIN {X 0,Y 199.211,Z 309.94,A -85,B 0,C 180,E1 -21675.933,E2 -21675.933} C_VEL
LIN {X 0,Y 197.987,Z 312.302,A -85,B 0,C 180,E1 -21677.459,E2 -21677.459} C_VEL
LIN {X 0,Y 194.412,Z 315.533,A -85,B 0,C 180,E1 -21679.99,E2 -21679.99} C_VEL
LIN {X 0,Y 191.585,Z 317.591,A -85,B 0,C 180,E1 -21682.12,E2 -21682.12} C_VEL
LIN {X 0,Y 190.331,Z 318.868,A -85,B 0,C 180,E1 -21683.823,E2 -21683.823} C_VEL
LIN {X 0,Y 190.193,Z 319.196,A -85,B 0,C 180,E1 -21684.408,E2 -21684.408} C_VEL
LIN {X 0,Y 190.156,Z 320.843,A -85,B 0,C 180,E1 -21687.883,E2 -21687.883} C_VEL
LIN {X 0,Y 190.265,Z 321.254,A -85,B 0,C 180,E1 -21690.001,E2 -21690.001} C_VEL
LIN {X 0,Y 190.12,Z 321.06,A -85,B 0,C 180,E1 -21693.548,E2 -21693.548} C_VEL
LIN {X 0,Y 190.279,Z 320.137,A -85,B 0,C 180,E1 -21696.363,E2 -21696.363} C_VEL
LIN {X 0,Y 191.031,Z 317.326,A -85,B 0,C 180,E1 -21700.601,E2 -21700.601} C_VEL
LIN {X 0,Y 192.089,Z 314.103,A -85,B 0,C 180,E1 -21703.758,E2 -21703.758} C_VEL
LIN {X 0,Y 193.745,Z 309.826,A -85,B 0,C 180,E1 -21706.87,E2 -21706.87} C_VEL
LIN {X 0,Y 196.324,Z 303.361,A -85,B 0,C 180,E1 -21710.428,E2 -21710.428} C_VEL
LIN {X 0,Y 198.857,Z 296.751,A -85,B 0,C 180,E1 -21713.236,E2 -21713.236} C_VEL
LIN {X 0,Y 201.688,Z 289.097,A -85,B 0,C 180,E1 -21715.821,E2 -21715.821} C_VEL
LIN {X 0,Y 204.808,Z 280.394,A -85,B 0,C 180,E1 -21718.153,E2 -21718.153} C_VEL
LIN {X 0,Y 205.919,Z 276.398,A -85,B 0,C 180,E1 -21719.1,E2 -21719.1} C_VEL
LIN {X 0,Y 206.319,Z 265.774,A -85,B 0,C 180,E1 -21721.615,E2 -21721.615} C_VEL
LIN {X 0,Y 205.779,Z 254.645,A -85,B 0,C 180,E1 -21723.943,E2 -21723.943} C_VEL
LIN {X 0,Y 204.325,Z 243.36,A -85,B 0,C 180,E1 -21726.067,E2 -21726.067} C_VEL
LIN {X 0,Y 201.848,Z 232.442,A -85,B 0,C 180,E1 -21728.013,E2 -21728.013} C_VEL
LIN {X 0,Y 198.584,Z 223.423,A -85,B 0,C 180,E1 -21729.683,E2 -21729.683} C_VEL
LIN {X 0,Y 196.186,Z 218.589,A -85,B 0,C 180,E1 -21730.681,E2 -21730.681} C_VEL
LIN {X 0,Y 194.682,Z 215.616,A -85,B 0,C 180,E1 -21731.295,E2 -21731.295} C_VEL
LIN {X 0,Y 194.402,Z 214.304,A -85,B 0,C 180,E1 -21731.487,E2 -21731.487} C_VEL
LIN {X 0,Y 193.828,Z 210.854,A -85,B 0,C 180,E1 -21736.456,E2 -21736.456} C_VEL
LIN {X 0,Y 193.478,Z 208.784,A -85,B 0,C 180,E1 -21739.71,E2 -21739.71} C_VEL
LIN {X 0,Y 193.056,Z 206.062,A -85,B 0,C 180,E1 -21744.376,E2 -21744.376} C_VEL
LIN {X 0,Y 192.584,Z 203.5,A -85,B 0,C 180,E1 -21749.276,E2 -21749.276} C_VEL
LIN {X 0,Y 192.645,Z 203.491,A -85,B 0,C 180,E1 -21751.689,E2 -21751.689} C_VEL
LIN {X 0,Y 192.707,Z 203.481,A -85,B 0,C 180,E1 -21756.349,E2 -21756.349} C_VEL
LIN {X 0,Y 192.774,Z 203.472,A -85,B 0,C 180,E1 -21761.413,E2 -21761.413} C_VEL
LIN {X 0,Y 192.757,Z 203.473,A -85,B 0,C 180,E1 -21765.214,E2 -21765.214} C_VEL
LIN {X 0,Y 192.937,Z 203.451,A -85,B 0,C 180,E1 -21769.567,E2 -21769.567} C_VEL
LIN {X 0,Y 192.973,Z 203.447,A -85,B 0,C 180,E1 -21773.728,E2 -21773.728} C_VEL
LIN {X 0,Y 193.249,Z 203.411,A -85,B 0,C 180,E1 -21777.916,E2 -21777.916} C_VEL
LIN {X 0,Y 193.422,Z 203.391,A -85,B 0,C 180,E1 -21780,E2 -21780} C_VEL
LIN {X 0,Y 193.275,Z 203.411,A -85,B 0,C 180,E1 -21782.084,E2 -21782.084} C_VEL
LIN {X 0,Y 193.018,Z 203.441,A -85,B 0,C 180,E1 -21788.375,E2 -21788.375} C_VEL
LIN {X 0,Y 192.787,Z 203.47,A -85,B 0,C 180,E1 -21792.635,E2 -21792.635} C_VEL
LIN {X 0,Y 192.745,Z 203.475,A -85,B 0,C 180,E1 -21796.96,E2 -21796.96} C_VEL
LIN {X 0,Y 192.625,Z 203.491,A -85,B 0,C 180,E1 -21801.399,E2 -21801.399} C_VEL
LIN {X 0,Y 192.649,Z 203.486,A -85,B 0,C 180,E1 -21804.22,E2 -21804.22} C_VEL
LIN {X 0,Y 192.638,Z 203.489,A -85,B 0,C 180,E1 -21808.89,E2 -21808.89} C_VEL
LIN {X 0,Y 192.592,Z 203.496,A -85,B 0,C 180,E1 -21813.188,E2 -21813.188} C_VEL
LIN {X 0,Y 192.546,Z 203.5,A -85,B 0,C 180,E1 -21818.354,E2 -21818.354} C_VEL
LIN {X 0,Y 192.555,Z 203.734,A -85,B 0,C 180,E1 -21819.965,E2 -21819.965} C_VEL
LIN {X 0,Y 192.819,Z 205.583,A -85,B 0,C 180,E1 -21823.831,E2 -21823.831} C_VEL
LIN {X 0,Y 193.02,Z 206.815,A -85,B 0,C 180,E1 -21826.229,E2 -21826.229} C_VEL
LIN {X 0,Y 194.13,Z 209.817,A -85,B 0,C 180,E1 -21826.768,E2 -21826.768} C_VEL
LIN {X 0,Y 195.765,Z 212.232,A -85,B 0,C 180,E1 -21827.389,E2 -21827.389} C_VEL
LIN {X 0,Y 199.41,Z 219.706,A -85,B 0,C 180,E1 -21829.017,E2 -21829.017} C_VEL
LIN {X 0,Y 202.801,Z 228.524,A -85,B 0,C 180,E1 -21830.843,E2 -21830.843} C_VEL
LIN {X 0,Y 205.459,Z 238.261,A -85,B 0,C 180,E1 -21832.837,E2 -21832.837} C_VEL
LIN {X 0,Y 207.41,Z 248.47,A -85,B 0,C 180,E1 -21835.032,E2 -21835.032} C_VEL
LIN {X 0,Y 208.339,Z 259.144,A -85,B 0,C 180,E1 -21837.495,E2 -21837.495} C_VEL
LIN {X 0,Y 208.403,Z 262.921,A -85,B 0,C 180,E1 -21838.427,E2 -21838.427} C_VEL
LIN {X 0,Y 205.177,Z 273.132,A -85,B 0,C 180,E1 -21840.784,E2 -21840.784} C_VEL
LIN {X 0,Y 202.244,Z 281.296,A -85,B 0,C 180,E1 -21843.145,E2 -21843.145} C_VEL
LIN {X 0,Y 199.061,Z 289.292,A -85,B 0,C 180,E1 -21846.046,E2 -21846.046} C_VEL
LIN {X 0,Y 196.477,Z 295.694,A -85,B 0,C 180,E1 -21849.041,E2 -21849.041} C_VEL
LIN {X 0,Y 194.44,Z 300.763,A -85,B 0,C 180,E1 -21852.107,E2 -21852.107} C_VEL
LIN {X 0,Y 192.668,Z 304.697,A -85,B 0,C 180,E1 -21855.206,E2 -21855.206} C_VEL
LIN {X 0,Y 191.883,Z 306.714,A -85,B 0,C 180,E1 -21857.305,E2 -21857.305} C_VEL
LIN {X 0,Y 190.741,Z 309.522,A -85,B 0,C 180,E1 -21861.524,E2 -21861.524} C_VEL
LIN {X 0,Y 190.435,Z 310.301,A -85,B 0,C 180,E1 -21863.643,E2 -21863.643} C_VEL
LIN {X 0,Y 190.279,Z 310.673,A -85,B 0,C 180,E1 -21865.763,E2 -21865.763} C_VEL
LIN {X 0,Y 190.247,Z 310.667,A -85,B 0,C 180,E1 -21867.882,E2 -21867.882} C_VEL
LIN {X 0,Y 190.301,Z 310.284,A -85,B 0,C 180,E1 -21869.999,E2 -21869.999} C_VEL
LIN {X 0,Y 190.451,Z 309.498,A -85,B 0,C 180,E1 -21872.113,E2 -21872.113} C_VEL
LIN {X 0,Y 190.732,Z 308.288,A -85,B 0,C 180,E1 -21874.225,E2 -21874.225} C_VEL
LIN {X 0,Y 191.485,Z 305.41,A -85,B 0,C 180,E1 -21877.699,E2 -21877.699} C_VEL
LIN {X 0,Y 192.876,Z 300.761,A -85,B 0,C 180,E1 -21881.559,E2 -21881.559} C_VEL
LIN {X 0,Y 194.47,Z 295.721,A -85,B 0,C 180,E1 -21884.651,E2 -21884.651} C_VEL
LIN {X 0,Y 196.648,Z 289.365,A -85,B 0,C 180,E1 -21887.682,E2 -21887.682} C_VEL
LIN {X 0,Y 199.294,Z 281.431,A -85,B 0,C 180,E1 -21890.646,E2 -21890.646} C_VEL
LIN {X 0,Y 201.792,Z 273.344,A -85,B 0,C 180,E1 -21893.064,E2 -21893.064} C_VEL
LIN {X 0,Y 204.492,Z 263.485,A -85,B 0,C 180,E1 -21895.439,E2 -21895.439} C_VEL
LIN {X 0,Y 205.671,Z 258.868,A -85,B 0,C 180,E1 -21896.37,E2 -21896.37} C_VEL
LIN {X 0,Y 205.303,Z 250.771,A -85,B 0,C 180,E1 -21898.139,E2 -21898.139} C_VEL
LIN {X 0,Y 203.913,Z 240.368,A -85,B 0,C 180,E1 -21900.229,E2 -21900.229} C_VEL
LIN {X 0,Y 201.195,Z 228.273,A -85,B 0,C 180,E1 -21902.448,E2 -21902.448} C_VEL
LIN {X 0,Y 197.398,Z 217.175,A -85,B 0,C 180,E1 -21904.402,E2 -21904.402} C_VEL
LIN {X 0,Y 194.251,Z 210.046,A -85,B 0,C 180,E1 -21905.658,E2 -21905.658} C_VEL
LIN {X 0,Y 193.024,Z 207.322,A -85,B 0,C 180,E1 -21906.127,E2 -21906.127} C_VEL
LIN {X 0,Y 192.853,Z 206.5,A -85,B 0,C 180,E1 -21906.274,E2 -21906.274} C_VEL
LIN {X 0,Y 192.547,Z 203.829,A -85,B 0,C 180,E1 -21911.066,E2 -21911.066} C_VEL
LIN {X 0,Y 192.538,Z 203.505,A -85,B 0,C 180,E1 -21913.905,E2 -21913.905} C_VEL
LIN {X 0,Y 192.592,Z 203.497,A -85,B 0,C 180,E1 -21916.866,E2 -21916.866} C_VEL
LIN {X 0,Y 192.588,Z 203.495,A -85,B 0,C 180,E1 -21921.656,E2 -21921.656} C_VEL
LIN {X 0,Y 192.595,Z 203.493,A -85,B 0,C 180,E1 -21927.057,E2 -21927.057} C_VEL
LIN {X 0,Y 192.646,Z 203.486,A -85,B 0,C 180,E1 -21931.688,E2 -21931.688} C_VEL
LIN {X 0,Y 192.699,Z 203.459,A -85,B 0,C 180,E1 -21936.347,E2 -21936.347} C_VEL
LIN {X 0,Y 192.766,Z 203.441,A -85,B 0,C 180,E1 -21941.411,E2 -21941.411} C_VEL
LIN {X 0,Y 192.84,Z 203.461,A -85,B 0,C 180,E1 -21947.369,E2 -21947.369} C_VEL
LIN {X 0,Y 193.066,Z 203.433,A -85,B 0,C 180,E1 -21951.627,E2 -21951.627} C_VEL
LIN {X 0,Y 193.241,Z 203.406,A -85,B 0,C 180,E1 -21957.915,E2 -21957.915} C_VEL
LIN {X 0,Y 193.415,Z 203.393,A -85,B 0,C 180,E1 -21960,E2 -21960} C_VEL
LIN {X 0,Y 193.267,Z 203.412,A -85,B 0,C 180,E1 -21962.084,E2 -21962.084} C_VEL
LIN {X 0,Y 193.041,Z 203.439,A -85,B 0,C 180,E1 -21968.373,E2 -21968.373} C_VEL
LIN {X 0,Y 192.787,Z 203.471,A -85,B 0,C 180,E1 -21972.634,E2 -21972.634} C_VEL
LIN {X 0,Y 192.765,Z 203.475,A -85,B 0,C 180,E1 -21978.588,E2 -21978.588} C_VEL
LIN {X 0,Y 192.655,Z 203.488,A -85,B 0,C 180,E1 -21984.23,E2 -21984.23} C_VEL
LIN {X 0,Y 192.633,Z 203.482,A -85,B 0,C 180,E1 -21988.893,E2 -21988.893} C_VEL
LIN {X 0,Y 192.584,Z 203.496,A -85,B 0,C 180,E1 -21993.188,E2 -21993.188} C_VEL
LIN {X 0,Y 192.654,Z 203.721,A -85,B 0,C 180,E1 -21996.182,E2 -21996.182} C_VEL
LIN {X 0,Y 193.155,Z 206.647,A -85,B 0,C 180,E1 -22000.914,E2 -22000.914} C_VEL
LIN {X 0,Y 193.482,Z 208.442,A -85,B 0,C 180,E1 -22003.642,E2 -22003.642} C_VEL
LIN {X 0,Y 193.946,Z 211.456,A -85,B 0,C 180,E1 -22007.931,E2 -22007.931} C_VEL
LIN {X 0,Y 194.212,Z 214.583,A -85,B 0,C 180,E1 -22012.082,E2 -22012.082} C_VEL
LIN {X 0,Y 195.328,Z 217.971,A -85,B 0,C 180,E1 -22012.564,E2 -22012.564} C_VEL
LIN {X 0,Y 197.304,Z 222.996,A -85,B 0,C 180,E1 -22013.354,E2 -22013.354} C_VEL
LIN {X 0,Y 199.97,Z 232.712,A -85,B 0,C 180,E1 -22014.799,E2 -22014.799} C_VEL
LIN {X 0,Y 202.095,Z 243.874,A -85,B 0,C 180,E1 -22016.576,E2 -22016.576} C_VEL
LIN {X 0,Y 203.27,Z 254.654,A -85,B 0,C 180,E1 -22018.467,E2 -22018.467} C_VEL
LIN {X 0,Y 203.559,Z 265.22,A -85,B 0,C 180,E1 -22020.549,E2 -22020.549} C_VEL
LIN {X 0,Y 203.076,Z 274.82,A -85,B 0,C 180,E1 -22022.71,E2 -22022.71} C_VEL
LIN {X 0,Y 200.16,Z 284.576,A -85,B 0,C 180,E1 -22025.084,E2 -22025.084} C_VEL
LIN {X 0,Y 197.512,Z 293.586,A -85,B 0,C 180,E1 -22027.892,E2 -22027.892} C_VEL
LIN {X 0,Y 194.921,Z 301.547,A -85,B 0,C 180,E1 -22031.068,E2 -22031.068} C_VEL
LIN {X 0,Y 192.953,Z 307.604,A -85,B 0,C 180,E1 -22034.149,E2 -22034.149} C_VEL
LIN {X 0,Y 191.602,Z 312.403,A -85,B 0,C 180,E1 -22037.289,E2 -22037.289} C_VEL
LIN {X 0,Y 190.742,Z 316.081,A -85,B 0,C 180,E1 -22040.458,E2 -22040.458} C_VEL
LIN {X 0,Y 190.193,Z 319.196,A -85,B 0,C 180,E1 -22044.408,E2 -22044.408} C_VEL
LIN {X 0,Y 189.417,Z 320.18,A -85,B 0,C 180,E1 -22046.156,E2 -22046.156} C_VEL
LIN {X 0,Y 187.794,Z 320.782,A -85,B 0,C 180,E1 -22047.887,E2 -22047.887} C_VEL
LIN {X 0,Y 184.111,Z 321.162,A -85,B 0,C 180,E1 -22051.411,E2 -22051.411} C_VEL
LIN {X 0,Y 183.102,Z 320.967,A -85,B 0,C 180,E1 -22053.255,E2 -22053.255} C_VEL
LIN {X 0,Y 183.026,Z 320.826,A -85,B 0,C 180,E1 -22053.879,E2 -22053.879} C_VEL
LIN {X 0,Y 183.212,Z 319.954,A -85,B 0,C 180,E1 -22056.609,E2 -22056.609} C_VEL
LIN {X 0,Y 183.512,Z 318.759,A -85,B 0,C 180,E1 -22058.813,E2 -22058.813} C_VEL
LIN {X 0,Y 184.351,Z 316.214,A -85,B 0,C 180,E1 -22062.104,E2 -22062.104} C_VEL
LIN {X 0,Y 185.639,Z 312.666,A -85,B 0,C 180,E1 -22065.368,E2 -22065.368} C_VEL
LIN {X 0,Y 187.652,Z 308.025,A -85,B 0,C 180,E1 -22068.563,E2 -22068.563} C_VEL
LIN {X 0,Y 190.626,Z 301.111,A -85,B 0,C 180,E1 -22072.161,E2 -22072.161} C_VEL
LIN {X 0,Y 193.551,Z 293.463,A -85,B 0,C 180,E1 -22075.254,E2 -22075.254} C_VEL
LIN {X 0,Y 196.559,Z 285.745,A -85,B 0,C 180,E1 -22077.698,E2 -22077.698} C_VEL
LIN {X 0,Y 199.269,Z 278.369,A -85,B 0,C 180,E1 -22079.588,E2 -22079.588} C_VEL
LIN {X 0,Y 199.92,Z 268.299,A -85,B 0,C 180,E1 -22082.156,E2 -22082.156} C_VEL
LIN {X 0,Y 199.719,Z 258,A -85,B 0,C 180,E1 -22084.472,E2 -22084.472} C_VEL
LIN {X 0,Y 198.51,Z 246.455,A -85,B 0,C 180,E1 -22086.815,E2 -22086.815} C_VEL
LIN {X 0,Y 196.22,Z 235.335,A -85,B 0,C 180,E1 -22088.959,E2 -22088.959} C_VEL
LIN {X 0,Y 193.112,Z 226.639,A -85,B 0,C 180,E1 -22090.762,E2 -22090.762} C_VEL
LIN {X 0,Y 190.834,Z 221.925,A -85,B 0,C 180,E1 -22091.827,E2 -22091.827} C_VEL
LIN {X 0,Y 189.28,Z 218.663,A -85,B 0,C 180,E1 -22092.538,E2 -22092.538} C_VEL
LIN {X 0,Y 187.539,Z 215.473,A -85,B 0,C 180,E1 -22093.299,E2 -22093.299} C_VEL
LIN {X 0,Y 187.176,Z 213.998,A -85,B 0,C 180,E1 -22093.582,E2 -22093.582} C_VEL
LIN {X 0,Y 186.574,Z 210.632,A -85,B 0,C 180,E1 -22098.881,E2 -22098.881} C_VEL
LIN {X 0,Y 186.24,Z 208.333,A -85,B 0,C 180,E1 -22102.859,E2 -22102.859} C_VEL
LIN {X 0,Y 185.79,Z 205.597,A -85,B 0,C 180,E1 -22108.023,E2 -22108.023} C_VEL
LIN {X 0,Y 185.572,Z 204.393,A -85,B 0,C 180,E1 -22110.577,E2 -22110.577} C_VEL
LIN {X 0,Y 185.6,Z 204.366,A -85,B 0,C 180,E1 -22115.385,E2 -22115.385} C_VEL
LIN {X 0,Y 185.704,Z 204.353,A -85,B 0,C 180,E1 -22121.1,E2 -22121.1} C_VEL
LIN {X 0,Y 185.692,Z 204.356,A -85,B 0,C 180,E1 -22124.637,E2 -22124.637} C_VEL
LIN {X 0,Y 185.88,Z 204.331,A -85,B 0,C 180,E1 -22129.418,E2 -22129.418} C_VEL
LIN {X 0,Y 185.936,Z 204.324,A -85,B 0,C 180,E1 -22133.489,E2 -22133.489} C_VEL
LIN {X 0,Y 186.193,Z 204.29,A -85,B 0,C 180,E1 -22137.837,E2 -22137.837} C_VEL
LIN {X 0,Y 186.387,Z 204.267,A -85,B 0,C 180,E1 -22140,E2 -22140} C_VEL
LIN {X 0,Y 185.922,Z 204.326,A -85,B 0,C 180,E1 -22144.336,E2 -22144.336} C_VEL
LIN {X 0,Y 185.967,Z 204.318,A -85,B 0,C 180,E1 -22148.695,E2 -22148.695} C_VEL
LIN {X 0,Y 185.715,Z 204.351,A -85,B 0,C 180,E1 -22153.125,E2 -22153.125} C_VEL
LIN {X 0,Y 185.68,Z 204.355,A -85,B 0,C 180,E1 -22157.627,E2 -22157.627} C_VEL
LIN {X 0,Y 185.584,Z 204.366,A -85,B 0,C 180,E1 -22162.254,E2 -22162.254} C_VEL
LIN {X 0,Y 185.553,Z 204.371,A -85,B 0,C 180,E1 -22167.034,E2 -22167.034} C_VEL
LIN {X 0,Y 185.573,Z 204.37,A -85,B 0,C 180,E1 -22169.495,E2 -22169.495} C_VEL
LIN {X 0,Y 185.494,Z 204.381,A -85,B 0,C 180,E1 -22174.634,E2 -22174.634} C_VEL
LIN {X 0,Y 185.501,Z 204.374,A -85,B 0,C 180,E1 -22177.315,E2 -22177.315} C_VEL
LIN {X 0,Y 185.668,Z 205.498,A -85,B 0,C 180,E1 -22180.798,E2 -22180.798} C_VEL
LIN {X 0,Y 185.857,Z 207.077,A -85,B 0,C 180,E1 -22184.147,E2 -22184.147} C_VEL
LIN {X 0,Y 187.046,Z 210.176,A -85,B 0,C 180,E1 -22184.775,E2 -22184.775} C_VEL
LIN {X 0,Y 188.684,Z 212.417,A -85,B 0,C 180,E1 -22185.445,E2 -22185.445} C_VEL
LIN {X 0,Y 190.84,Z 216.364,A -85,B 0,C 180,E1 -22186.439,E2 -22186.439} C_VEL
LIN {X 0,Y 194.379,Z 223.915,A -85,B 0,C 180,E1 -22188.222,E2 -22188.222} C_VEL
LIN {X 0,Y 197.415,Z 232.482,A -85,B 0,C 180,E1 -22190.15,E2 -22190.15} C_VEL
LIN {X 0,Y 199.965,Z 242.967,A -85,B 0,C 180,E1 -22192.472,E2 -22192.472} C_VEL
LIN {X 0,Y 201.4,Z 252.361,A -85,B 0,C 180,E1 -22194.655,E2 -22194.655} C_VEL
LIN {X 0,Y 201.948,Z 261.69,A -85,B 0,C 180,E1 -22196.973,E2 -22196.973} C_VEL
LIN {X 0,Y 201.894,Z 264.65,A -85,B 0,C 180,E1 -22197.747,E2 -22197.747} C_VEL
LIN {X 0,Y 198.339,Z 274.98,A -85,B 0,C 180,E1 -22200.26,E2 -22200.26} C_VEL
LIN {X 0,Y 195.319,Z 282.868,A -85,B 0,C 180,E1 -22202.693,E2 -22202.693} C_VEL
LIN {X 0,Y 192.056,Z 290.571,A -85,B 0,C 180,E1 -22205.69,E2 -22205.69} C_VEL
LIN {X 0,Y 189.836,Z 295.823,A -85,B 0,C 180,E1 -22208.271,E2 -22208.271} C_VEL
LIN {X 0,Y 187.671,Z 300.909,A -85,B 0,C 180,E1 -22211.439,E2 -22211.439} C_VEL
LIN {X 0,Y 185.773,Z 304.856,A -85,B 0,C 180,E1 -22214.644,E2 -22214.644} C_VEL
LIN {X 0,Y 184.919,Z 306.88,A -85,B 0,C 180,E1 -22216.818,E2 -22216.818} C_VEL
LIN {X 0,Y 183.721,Z 309.699,A -85,B 0,C 180,E1 -22221.197,E2 -22221.197} C_VEL
LIN {X 0,Y 183.379,Z 310.49,A -85,B 0,C 180,E1 -22223.397,E2 -22223.397} C_VEL
LIN {X 0,Y 183.157,Z 310.868,A -85,B 0,C 180,E1 -22227.8,E2 -22227.8} C_VEL
LIN {X 0,Y 183.206,Z 310.491,A -85,B 0,C 180,E1 -22229.999,E2 -22229.999} C_VEL
LIN {X 0,Y 183.363,Z 309.715,A -85,B 0,C 180,E1 -22232.195,E2 -22232.195} C_VEL
LIN {X 0,Y 183.659,Z 308.512,A -85,B 0,C 180,E1 -22234.388,E2 -22234.388} C_VEL
LIN {X 0,Y 184.378,Z 305.966,A -85,B 0,C 180,E1 -22237.664,E2 -22237.664} C_VEL
LIN {X 0,Y 185.449,Z 302.424,A -85,B 0,C 180,E1 -22240.921,E2 -22240.921} C_VEL
LIN {X 0,Y 187,Z 297.782,A -85,B 0,C 180,E1 -22244.137,E2 -22244.137} C_VEL
LIN {X 0,Y 189.485,Z 290.789,A -85,B 0,C 180,E1 -22247.815,E2 -22247.815} C_VEL
LIN {X 0,Y 192.18,Z 283.207,A -85,B 0,C 180,E1 -22250.886,E2 -22250.886} C_VEL
LIN {X 0,Y 194.673,Z 275.446,A -85,B 0,C 180,E1 -22253.395,E2 -22253.395} C_VEL
LIN {X 0,Y 197.83,Z 264.901,A -85,B 0,C 180,E1 -22256.077,E2 -22256.077} C_VEL
LIN {X 0,Y 199.201,Z 259.245,A -85,B 0,C 180,E1 -22257.297,E2 -22257.297} C_VEL
LIN {X 0,Y 198.531,Z 248.685,A -85,B 0,C 180,E1 -22259.705,E2 -22259.705} C_VEL
LIN {X 0,Y 197.084,Z 239.461,A -85,B 0,C 180,E1 -22261.637,E2 -22261.637} C_VEL
LIN {X 0,Y 194.514,Z 228.208,A -85,B 0,C 180,E1 -22263.795,E2 -22263.795} C_VEL
LIN {X 0,Y 190.622,Z 217.383,A -85,B 0,C 180,E1 -22265.866,E2 -22265.866} C_VEL
LIN {X 0,Y 187.465,Z 210.721,A -85,B 0,C 180,E1 -22267.186,E2 -22267.186} C_VEL
LIN {X 0,Y 185.998,Z 207.835,A -85,B 0,C 180,E1 -22267.767,E2 -22267.767} C_VEL
LIN {X 0,Y 185.764,Z 206.75,A -85,B 0,C 180,E1 -22267.954,E2 -22267.954} C_VEL
LIN {X 0,Y 185.589,Z 205.243,A -85,B 0,C 180,E1 -22270.766,E2 -22270.766} C_VEL
LIN {X 0,Y 185.489,Z 204.383,A -85,B 0,C 180,E1 -22272.994,E2 -22272.994} C_VEL
LIN {X 0,Y 185.545,Z 204.376,A -85,B 0,C 180,E1 -22277.015,E2 -22277.015} C_VEL
LIN {X 0,Y 185.532,Z 204.374,A -85,B 0,C 180,E1 -22279.911,E2 -22279.911} C_VEL
LIN {X 0,Y 185.534,Z 204.373,A -85,B 0,C 180,E1 -22282.693,E2 -22282.693} C_VEL
LIN {X 0,Y 185.529,Z 204.371,A -85,B 0,C 180,E1 -22287.971,E2 -22287.971} C_VEL
LIN {X 0,Y 185.568,Z 204.368,A -85,B 0,C 180,E1 -22290.574,E2 -22290.574} C_VEL
LIN {X 0,Y 185.592,Z 204.354,A -85,B 0,C 180,E1 -22295.382,E2 -22295.382} C_VEL
LIN {X 0,Y 185.696,Z 204.315,A -85,B 0,C 180,E1 -22301.099,E2 -22301.099} C_VEL
LIN {X 0,Y 185.715,Z 204.35,A -85,B 0,C 180,E1 -22304.638,E2 -22304.638} C_VEL
LIN {X 0,Y 185.926,Z 204.31,A -85,B 0,C 180,E1 -22309.327,E2 -22309.327} C_VEL
LIN {X 0,Y 185.951,Z 204.322,A -85,B 0,C 180,E1 -22313.489,E2 -22313.489} C_VEL
LIN {X 0,Y 186.186,Z 204.284,A -85,B 0,C 180,E1 -22317.836,E2 -22317.836} C_VEL
LIN {X 0,Y 186.38,Z 204.27,A -85,B 0,C 180,E1 -22320,E2 -22320} C_VEL
LIN {X 0,Y 185.919,Z 204.326,A -85,B 0,C 180,E1 -22324.335,E2 -22324.335} C_VEL
LIN {X 0,Y 185.989,Z 204.318,A -85,B 0,C 180,E1 -22328.693,E2 -22328.693} C_VEL
LIN {X 0,Y 185.711,Z 204.355,A -85,B 0,C 180,E1 -22333.124,E2 -22333.124} C_VEL
LIN {X 0,Y 185.695,Z 204.355,A -85,B 0,C 180,E1 -22338.9,E2 -22338.9} C_VEL
LIN {X 0,Y 185.591,Z 204.367,A -85,B 0,C 180,E1 -22344.617,E2 -22344.617} C_VEL
LIN {X 0,Y 185.564,Z 204.355,A -85,B 0,C 180,E1 -22349.495,E2 -22349.495} C_VEL
LIN {X 0,Y 185.52,Z 204.449,A -85,B 0,C 180,E1 -22354.958,E2 -22354.958} C_VEL
LIN {X 0,Y 186.053,Z 207.341,A -85,B 0,C 180,E1 -22359.953,E2 -22359.953} C_VEL
LIN {X 0,Y 186.54,Z 210.093,A -85,B 0,C 180,E1 -22364.295,E2 -22364.295} C_VEL
LIN {X 0,Y 187.029,Z 213.126,A -85,B 0,C 180,E1 -22368.724,E2 -22368.724} C_VEL
LIN {X 0,Y 187.108,Z 214.504,A -85,B 0,C 180,E1 -22370.458,E2 -22370.458} C_VEL
LIN {X 0,Y 188.253,Z 217.76,A -85,B 0,C 180,E1 -22370.956,E2 -22370.956} C_VEL
LIN {X 0,Y 189.379,Z 219.995,A -85,B 0,C 180,E1 -22371.384,E2 -22371.384} C_VEL
LIN {X 0,Y 191.838,Z 226.536,A -85,B 0,C 180,E1 -22372.504,E2 -22372.504} C_VEL
LIN {X 0,Y 194.591,Z 237.842,A -85,B 0,C 180,E1 -22374.355,E2 -22374.355} C_VEL
LIN {X 0,Y 196.316,Z 249.429,A -85,B 0,C 180,E1 -22376.391,E2 -22376.391} C_VEL
LIN {X 0,Y 197.062,Z 259.735,A -85,B 0,C 180,E1 -22378.403,E2 -22378.403} C_VEL
LIN {X 0,Y 196.888,Z 269.857,A -85,B 0,C 180,E1 -22380.61,E2 -22380.61} C_VEL
LIN {X 0,Y 196.45,Z 275.555,A -85,B 0,C 180,E1 -22381.999,E2 -22381.999} C_VEL
LIN {X 0,Y 193.719,Z 284.262,A -85,B 0,C 180,E1 -22384.196,E2 -22384.196} C_VEL
LIN {X 0,Y 191.043,Z 292.735,A -85,B 0,C 180,E1 -22386.88,E2 -22386.88} C_VEL
LIN {X 0,Y 188.563,Z 300.151,A -85,B 0,C 180,E1 -22389.836,E2 -22389.836} C_VEL
LIN {X 0,Y 186.763,Z 305.495,A -85,B 0,C 180,E1 -22392.482,E2 -22392.482} C_VEL
LIN {X 0,Y 185.042,Z 310.708,A -85,B 0,C 180,E1 -22395.71,E2 -22395.71} C_VEL
LIN {X 0,Y 183.964,Z 314.759,A -85,B 0,C 180,E1 -22398.99,E2 -22398.99} C_VEL
LIN {X 0,Y 183.508,Z 316.855,A -85,B 0,C 180,E1 -22401.19,E2 -22401.19} C_VEL
LIN {X 0,Y 183.101,Z 319.07,A -85,B 0,C 180,E1 -22404.357,E2 -22404.357} C_VEL
LIN {X 0,Y 183.051,Z 320.635,A -85,B 0,C 180,E1 -22407.801,E2 -22407.801} C_VEL
LIN {X 0,Y 183.17,Z 321.054,A -85,B 0,C 180,E1 -22410.001,E2 -22410.001} C_VEL
LIN {X 0,Y 183.026,Z 320.826,A -85,B 0,C 180,E1 -22413.879,E2 -22413.879} C_VEL
LIN {X 0,Y 182.431,Z 320.295,A -85,B 0,C 180,E1 -22415.712,E2 -22415.712} C_VEL
LIN {X 0,Y 179.944,Z 318.851,A -85,B 0,C 180,E1 -22418.712,E2 -22418.712} C_VEL
LIN {X 0,Y 178.074,Z 317.204,A -85,B 0,C 180,E1 -22421.138,E2 -22421.138} C_VEL
LIN {X 0,Y 177.613,Z 315.68,A -85,B 0,C 180,E1 -22422.982,E2 -22422.982} C_VEL
LIN {X 0,Y 177.754,Z 315.097,A -85,B 0,C 180,E1 -22423.592,E2 -22423.592} C_VEL
LIN {X 0,Y 179.433,Z 311.081,A -85,B 0,C 180,E1 -22427.083,E2 -22427.083} C_VEL
LIN {X 0,Y 181.706,Z 306.067,A -85,B 0,C 180,E1 -22430.371,E2 -22430.371} C_VEL
LIN {X 0,Y 184.492,Z 299.966,A -85,B 0,C 180,E1 -22433.479,E2 -22433.479} C_VEL
LIN {X 0,Y 187.127,Z 293.351,A -85,B 0,C 180,E1 -22436.186,E2 -22436.186} C_VEL
LIN {X 0,Y 190.282,Z 285.653,A -85,B 0,C 180,E1 -22438.695,E2 -22438.695} C_VEL
LIN {X 0,Y 192.384,Z 280.251,A -85,B 0,C 180,E1 -22440.152,E2 -22440.152} C_VEL
LIN {X 0,Y 193.178,Z 275.202,A -85,B 0,C 180,E1 -22441.531,E2 -22441.531} C_VEL
LIN {X 0,Y 193.624,Z 266.266,A -85,B 0,C 180,E1 -22443.823,E2 -22443.823} C_VEL
LIN {X 0,Y 193.318,Z 256.943,A -85,B 0,C 180,E1 -22446.002,E2 -22446.002} C_VEL
LIN {X 0,Y 192.252,Z 246.716,A -85,B 0,C 180,E1 -22448.193,E2 -22448.193} C_VEL
LIN {X 0,Y 190.667,Z 238.454,A -85,B 0,C 180,E1 -22449.904,E2 -22449.904} C_VEL
LIN {X 0,Y 187.921,Z 230.396,A -85,B 0,C 180,E1 -22451.719,E2 -22451.719} C_VEL
LIN {X 0,Y 184.625,Z 223.206,A -85,B 0,C 180,E1 -22453.478,E2 -22453.478} C_VEL
LIN {X 0,Y 182.335,Z 218.732,A -85,B 0,C 180,E1 -22454.616,E2 -22454.616} C_VEL
LIN {X 0,Y 180.454,Z 215.681,A -85,B 0,C 180,E1 -22455.49,E2 -22455.49} C_VEL
LIN {X 0,Y 179.888,Z 213.736,A -85,B 0,C 180,E1 -22455.886,E2 -22455.886} C_VEL
LIN {X 0,Y 179.368,Z 210.672,A -85,B 0,C 180,E1 -22461.178,E2 -22461.178} C_VEL
LIN {X 0,Y 178.924,Z 207.765,A -85,B 0,C 180,E1 -22466.64,E2 -22466.64} C_VEL
LIN {X 0,Y 178.503,Z 205.409,A -85,B 0,C 180,E1 -22471.806,E2 -22471.806} C_VEL
LIN {X 0,Y 178.526,Z 205.247,A -85,B 0,C 180,E1 -22476.817,E2 -22476.817} C_VEL
LIN {X 0,Y 178.673,Z 205.229,A -85,B 0,C 180,E1 -22481.659,E2 -22481.659} C_VEL
LIN {X 0,Y 178.65,Z 205.232,A -85,B 0,C 180,E1 -22486.348,E2 -22486.348} C_VEL
LIN {X 0,Y 178.902,Z 205.201,A -85,B 0,C 180,E1 -22490.96,E2 -22490.96} C_VEL
LIN {X 0,Y 179.139,Z 205.169,A -85,B 0,C 180,E1 -22497.752,E2 -22497.752} C_VEL
LIN {X 0,Y 179.352,Z 205.143,A -85,B 0,C 180,E1 -22500.001,E2 -22500.001} C_VEL
LIN {X 0,Y 178.868,Z 205.205,A -85,B 0,C 180,E1 -22504.508,E2 -22504.508} C_VEL
LIN {X 0,Y 178.898,Z 205.198,A -85,B 0,C 180,E1 -22509.042,E2 -22509.042} C_VEL
LIN {X 0,Y 178.644,Z 205.233,A -85,B 0,C 180,E1 -22513.654,E2 -22513.654} C_VEL
LIN {X 0,Y 178.616,Z 205.236,A -85,B 0,C 180,E1 -22519.216,E2 -22519.216} C_VEL
LIN {X 0,Y 178.515,Z 205.248,A -85,B 0,C 180,E1 -22525.116,E2 -22525.116} C_VEL
LIN {X 0,Y 178.517,Z 205.248,A -85,B 0,C 180,E1 -22529.994,E2 -22529.994} C_VEL
LIN {X 0,Y 178.48,Z 205.254,A -85,B 0,C 180,E1 -22534.22,E2 -22534.22} C_VEL
LIN {X 0,Y 178.418,Z 205.261,A -85,B 0,C 180,E1 -22536.219,E2 -22536.219} C_VEL
LIN {X 0,Y 178.537,Z 206.141,A -85,B 0,C 180,E1 -22539.039,E2 -22539.039} C_VEL
LIN {X 0,Y 178.76,Z 207.456,A -85,B 0,C 180,E1 -22541.867,E2 -22541.867} C_VEL
LIN {X 0,Y 179.964,Z 210.466,A -85,B 0,C 180,E1 -22542.54,E2 -22542.54} C_VEL
LIN {X 0,Y 181.863,Z 213.129,A -85,B 0,C 180,E1 -22543.406,E2 -22543.406} C_VEL
LIN {X 0,Y 183.906,Z 216.774,A -85,B 0,C 180,E1 -22544.439,E2 -22544.439} C_VEL
LIN {X 0,Y 187.308,Z 223.483,A -85,B 0,C 180,E1 -22546.244,E2 -22546.244} C_VEL
LIN {X 0,Y 190.778,Z 232.323,A -85,B 0,C 180,E1 -22548.466,E2 -22548.466} C_VEL
LIN {X 0,Y 193.123,Z 241.016,A -85,B 0,C 180,E1 -22550.538,E2 -22550.538} C_VEL
LIN {X 0,Y 194.811,Z 250.98,A -85,B 0,C 180,E1 -22552.958,E2 -22552.958} C_VEL
LIN {X 0,Y 195.534,Z 260.104,A -85,B 0,C 180,E1 -22555.313,E2 -22555.313} C_VEL
LIN {X 0,Y 195.354,Z 266.375,A -85,B 0,C 180,E1 -22557.014,E2 -22557.014} C_VEL
LIN {X 0,Y 192.194,Z 275.048,A -85,B 0,C 180,E1 -22559.208,E2 -22559.208} C_VEL
LIN {X 0,Y 189.029,Z 282.958,A -85,B 0,C 180,E1 -22561.704,E2 -22561.704} C_VEL
LIN {X 0,Y 185.573,Z 290.688,A -85,B 0,C 180,E1 -22564.783,E2 -22564.783} C_VEL
LIN {X 0,Y 183.237,Z 295.951,A -85,B 0,C 180,E1 -22567.447,E2 -22567.447} C_VEL
LIN {X 0,Y 180.919,Z 301.054,A -85,B 0,C 180,E1 -22570.719,E2 -22570.719} C_VEL
LIN {X 0,Y 178.903,Z 305.014,A -85,B 0,C 180,E1 -22574.038,E2 -22574.038} C_VEL
LIN {X 0,Y 177.98,Z 307.046,A -85,B 0,C 180,E1 -22576.294,E2 -22576.294} C_VEL
LIN {X 0,Y 176.694,Z 309.877,A -85,B 0,C 180,E1 -22580.844,E2 -22580.844} C_VEL
LIN {X 0,Y 176.324,Z 310.679,A -85,B 0,C 180,E1 -22583.131,E2 -22583.131} C_VEL
LIN {X 0,Y 176.086,Z 311.116,A -85,B 0,C 180,E1 -22586.22,E2 -22586.22} C_VEL
LIN {X 0,Y 176.114,Z 310.697,A -85,B 0,C 180,E1 -22589.998,E2 -22589.998} C_VEL
LIN {X 0,Y 176.277,Z 309.932,A -85,B 0,C 180,E1 -22592.283,E2 -22592.283} C_VEL
LIN {X 0,Y 176.589,Z 308.736,A -85,B 0,C 180,E1 -22594.564,E2 -22594.564} C_VEL
LIN {X 0,Y 177.225,Z 306.613,A -85,B 0,C 180,E1 -22597.516,E2 -22597.516} C_VEL
LIN {X 0,Y 178.48,Z 302.673,A -85,B 0,C 180,E1 -22601.352,E2 -22601.352} C_VEL
LIN {X 0,Y 180.138,Z 298.045,A -85,B 0,C 180,E1 -22604.688,E2 -22604.688} C_VEL
LIN {X 0,Y 182.737,Z 291.068,A -85,B 0,C 180,E1 -22608.496,E2 -22608.496} C_VEL
LIN {X 0,Y 185.582,Z 283.507,A -85,B 0,C 180,E1 -22611.665,E2 -22611.665} C_VEL
LIN {X 0,Y 188.185,Z 275.77,A -85,B 0,C 180,E1 -22614.252,E2 -22614.252} C_VEL
LIN {X 0,Y 191.492,Z 265.253,A -85,B 0,C 180,E1 -22617.008,E2 -22617.008} C_VEL
LIN {X 0,Y 192.701,Z 260.775,A -85,B 0,C 180,E1 -22618.002,E2 -22618.002} C_VEL
LIN {X 0,Y 192.209,Z 250.688,A -85,B 0,C 180,E1 -22620.452,E2 -22620.452} C_VEL
LIN {X 0,Y 190.791,Z 240.963,A -85,B 0,C 180,E1 -22622.623,E2 -22622.623} C_VEL
LIN {X 0,Y 188.813,Z 231.565,A -85,B 0,C 180,E1 -22624.558,E2 -22624.558} C_VEL
LIN {X 0,Y 185.059,Z 220.588,A -85,B 0,C 180,E1 -22626.845,E2 -22626.845} C_VEL
LIN {X 0,Y 181.891,Z 213.895,A -85,B 0,C 180,E1 -22628.332,E2 -22628.332} C_VEL
LIN {X 0,Y 180.437,Z 210.998,A -85,B 0,C 180,E1 -22628.963,E2 -22628.963} C_VEL
LIN {X 0,Y 178.927,Z 208.071,A -85,B 0,C 180,E1 -22629.613,E2 -22629.613} C_VEL
LIN {X 0,Y 178.678,Z 206.972,A -85,B 0,C 180,E1 -22629.825,E2 -22629.825} C_VEL
LIN {X 0,Y 178.502,Z 205.892,A -85,B 0,C 180,E1 -22632.009,E2 -22632.009} C_VEL
LIN {X 0,Y 178.453,Z 205.255,A -85,B 0,C 180,E1 -22635.138,E2 -22635.138} C_VEL
LIN {X 0,Y 178.493,Z 205.252,A -85,B 0,C 180,E1 -22638.42,E2 -22638.42} C_VEL
LIN {X 0,Y 178.436,Z 205.258,A -85,B 0,C 180,E1 -22643.785,E2 -22643.785} C_VEL
LIN {X 0,Y 178.475,Z 205.255,A -85,B 0,C 180,E1 -22646.543,E2 -22646.543} C_VEL
LIN {X 0,Y 178.509,Z 205.249,A -85,B 0,C 180,E1 -22650.004,E2 -22650.004} C_VEL
LIN {X 0,Y 178.521,Z 205.24,A -85,B 0,C 180,E1 -22654.873,E2 -22654.873} C_VEL
LIN {X 0,Y 178.64,Z 205.187,A -85,B 0,C 180,E1 -22660.753,E2 -22660.753} C_VEL
LIN {X 0,Y 178.662,Z 205.224,A -85,B 0,C 180,E1 -22664.016,E2 -22664.016} C_VEL
LIN {X 0,Y 178.879,Z 205.187,A -85,B 0,C 180,E1 -22669.152,E2 -22669.152} C_VEL
LIN {X 0,Y 178.917,Z 205.198,A -85,B 0,C 180,E1 -22673.232,E2 -22673.232} C_VEL
LIN {X 0,Y 179.132,Z 205.162,A -85,B 0,C 180,E1 -22677.751,E2 -22677.751} C_VEL
LIN {X 0,Y 179.344,Z 205.146,A -85,B 0,C 180,E1 -22679.999,E2 -22679.999} C_VEL
LIN {X 0,Y 178.866,Z 205.204,A -85,B 0,C 180,E1 -22684.507,E2 -22684.507} C_VEL
LIN {X 0,Y 178.94,Z 205.196,A -85,B 0,C 180,E1 -22689.038,E2 -22689.038} C_VEL
LIN {X 0,Y 178.639,Z 205.234,A -85,B 0,C 180,E1 -22693.653,E2 -22693.653} C_VEL
LIN {X 0,Y 178.639,Z 205.235,A -85,B 0,C 180,E1 -22699.246,E2 -22699.246} C_VEL
LIN {X 0,Y 178.52,Z 205.248,A -85,B 0,C 180,E1 -22705.126,E2 -22705.126} C_VEL
LIN {X 0,Y 178.508,Z 205.23,A -85,B 0,C 180,E1 -22709.995,E2 -22709.995} C_VEL
LIN {X 0,Y 178.501,Z 205.367,A -85,B 0,C 180,E1 -22714.016,E2 -22714.016} C_VEL
LIN {X 0,Y 178.87,Z 207.643,A -85,B 0,C 180,E1 -22718.211,E2 -22718.211} C_VEL
LIN {X 0,Y 179.255,Z 209.784,A -85,B 0,C 180,E1 -22721.854,E2 -22721.854} C_VEL
LIN {X 0,Y 179.625,Z 211.893,A -85,B 0,C 180,E1 -22725.236,E2 -22725.236} C_VEL
LIN {X 0,Y 180.055,Z 214.344,A -85,B 0,C 180,E1 -22728.648,E2 -22728.648} C_VEL
LIN {X 0,Y 181.08,Z 217.375,A -85,B 0,C 180,E1 -22729.143,E2 -22729.143} C_VEL
LIN {X 0,Y 182.333,Z 219.713,A -85,B 0,C 180,E1 -22729.651,E2 -22729.651} C_VEL
LIN {X 0,Y 185.734,Z 227.958,A -85,B 0,C 180,E1 -22731.271,E2 -22731.271} C_VEL
LIN {X 0,Y 188.222,Z 237.976,A -85,B 0,C 180,E1 -22733.049,E2 -22733.049} C_VEL
LIN {X 0,Y 189.976,Z 250.201,A -85,B 0,C 180,E1 -22735.332,E2 -22735.332} C_VEL
LIN {X 0,Y 190.622,Z 260.777,A -85,B 0,C 180,E1 -22737.518,E2 -22737.518} C_VEL
LIN {X 0,Y 190.359,Z 270.684,A -85,B 0,C 180,E1 -22739.803,E2 -22739.803} C_VEL
LIN {X 0,Y 189.871,Z 276.292,A -85,B 0,C 180,E1 -22741.241,E2 -22741.241} C_VEL
LIN {X 0,Y 186.753,Z 285.706,A -85,B 0,C 180,E1 -22743.76,E2 -22743.76} C_VEL
LIN {X 0,Y 183.901,Z 294.304,A -85,B 0,C 180,E1 -22746.725,E2 -22746.725} C_VEL
LIN {X 0,Y 181.092,Z 302.128,A -85,B 0,C 180,E1 -22750.152,E2 -22750.152} C_VEL
LIN {X 0,Y 179.292,Z 307.089,A -85,B 0,C 180,E1 -22752.906,E2 -22752.906} C_VEL
LIN {X 0,Y 177.7,Z 311.912,A -85,B 0,C 180,E1 -22756.275,E2 -22756.275} C_VEL
LIN {X 0,Y 176.693,Z 315.614,A -85,B 0,C 180,E1 -22759.691,E2 -22759.691} C_VEL
LIN {X 0,Y 176.138,Z 318.298,A -85,B 0,C 180,E1 -22763.127,E2 -22763.127} C_VEL
LIN {X 0,Y 175.92,Z 320.229,A -85,B 0,C 180,E1 -22767.129,E2 -22767.129} C_VEL
LIN {X 0,Y 176.077,Z 320.854,A -85,B 0,C 180,E1 -22770.002,E2 -22770.002} C_VEL
LIN {X 0,Y 175.933,Z 320.656,A -85,B 0,C 180,E1 -22773.88,E2 -22773.88} C_VEL
LIN {X 0,Y 176.14,Z 319.771,A -85,B 0,C 180,E1 -22776.876,E2 -22776.876} C_VEL
LIN {X 0,Y 176.475,Z 318.584,A -85,B 0,C 180,E1 -22779.167,E2 -22779.167} C_VEL
LIN {X 0,Y 177.754,Z 315.097,A -85,B 0,C 180,E1 -22783.592,E2 -22783.592} C_VEL
LIN {X 0,Y 177.856,Z 313.272,A -85,B 0,C 180,E1 -22785.407,E2 -22785.407} C_VEL
LIN {X 0,Y 176.602,Z 309.81,A -85,B 0,C 180,E1 -22788.392,E2 -22788.392} C_VEL
LIN {X 0,Y 175.81,Z 305.652,A -85,B 0,C 180,E1 -22791.309,E2 -22791.309} C_VEL
LIN {X 0,Y 176.612,Z 302.739,A -85,B 0,C 180,E1 -22792.959,E2 -22792.959} C_VEL
LIN {X 0,Y 179.602,Z 295.955,A -85,B 0,C 180,E1 -22796.118,E2 -22796.118} C_VEL
LIN {X 0,Y 183.386,Z 287.191,A -85,B 0,C 180,E1 -22799.25,E2 -22799.25} C_VEL
LIN {X 0,Y 186.189,Z 280.18,A -85,B 0,C 180,E1 -22801.265,E2 -22801.265} C_VEL
LIN {X 0,Y 187.172,Z 271.527,A -85,B 0,C 180,E1 -22803.728,E2 -22803.728} C_VEL
LIN {X 0,Y 187.342,Z 261.848,A -85,B 0,C 180,E1 -22806.215,E2 -22806.215} C_VEL
LIN {X 0,Y 186.704,Z 251.483,A -85,B 0,C 180,E1 -22808.642,E2 -22808.642} C_VEL
LIN {X 0,Y 185.327,Z 242.451,A -85,B 0,C 180,E1 -22810.673,E2 -22810.673} C_VEL
LIN {X 0,Y 182.922,Z 234.602,A -85,B 0,C 180,E1 -22812.571,E2 -22812.571} C_VEL
LIN {X 0,Y 179.607,Z 227.029,A -85,B 0,C 180,E1 -22814.609,E2 -22814.609} C_VEL
LIN {X 0,Y 177.898,Z 223.544,A -85,B 0,C 180,E1 -22815.574,E2 -22815.574} C_VEL
LIN {X 0,Y 175.931,Z 219.692,A -85,B 0,C 180,E1 -22816.672,E2 -22816.672} C_VEL
LIN {X 0,Y 174.484,Z 217.699,A -85,B 0,C 180,E1 -22817.377,E2 -22817.377} C_VEL
LIN {X 0,Y 172.895,Z 214.501,A -85,B 0,C 180,E1 -22818.271,E2 -22818.271} C_VEL
LIN {X 0,Y 172.636,Z 213.526,A -85,B 0,C 180,E1 -22818.454,E2 -22818.454} C_VEL
LIN {X 0,Y 172.285,Z 211.434,A -85,B 0,C 180,E1 -22822.274,E2 -22822.274} C_VEL
LIN {X 0,Y 172.078,Z 209.964,A -85,B 0,C 180,E1 -22825.126,E2 -22825.126} C_VEL
LIN {X 0,Y 171.654,Z 207.473,A -85,B 0,C 180,E1 -22830.573,E2 -22830.573} C_VEL
LIN {X 0,Y 171.461,Z 206.128,A -85,B 0,C 180,E1 -22834.385,E2 -22834.385} C_VEL
LIN {X 0,Y 171.604,Z 206.109,A -85,B 0,C 180,E1 -22840.875,E2 -22840.875} C_VEL
LIN {X 0,Y 171.571,Z 206.112,A -85,B 0,C 180,E1 -22845.773,E2 -22845.773} C_VEL
LIN {X 0,Y 171.839,Z 206.079,A -85,B 0,C 180,E1 -22850.585,E2 -22850.585} C_VEL
LIN {X 0,Y 171.801,Z 206.082,A -85,B 0,C 180,E1 -22855.308,E2 -22855.308} C_VEL
LIN {X 0,Y 172.316,Z 206.02,A -85,B 0,C 180,E1 -22860.001,E2 -22860.001} C_VEL
LIN {X 0,Y 171.815,Z 206.084,A -85,B 0,C 180,E1 -22864.693,E2 -22864.693} C_VEL
LIN {X 0,Y 171.836,Z 206.078,A -85,B 0,C 180,E1 -22869.416,E2 -22869.416} C_VEL
LIN {X 0,Y 171.562,Z 206.113,A -85,B 0,C 180,E1 -22874.229,E2 -22874.229} C_VEL
LIN {X 0,Y 171.537,Z 206.116,A -85,B 0,C 180,E1 -22879.561,E2 -22879.561} C_VEL
LIN {X 0,Y 171.453,Z 206.128,A -85,B 0,C 180,E1 -22885.61,E2 -22885.61} C_VEL
LIN {X 0,Y 171.435,Z 206.13,A -85,B 0,C 180,E1 -22890.586,E2 -22890.586} C_VEL
LIN {X 0,Y 171.389,Z 206.136,A -85,B 0,C 180,E1 -22895.036,E2 -22895.036} C_VEL
LIN {X 0,Y 171.577,Z 207.626,A -85,B 0,C 180,E1 -22899.207,E2 -22899.207} C_VEL
LIN {X 0,Y 172.68,Z 210.5,A -85,B 0,C 180,E1 -22899.909,E2 -22899.909} C_VEL
LIN {X 0,Y 174.884,Z 213.384,A -85,B 0,C 180,E1 -22901.019,E2 -22901.019} C_VEL
LIN {X 0,Y 176.802,Z 216.878,A -85,B 0,C 180,E1 -22902.106,E2 -22902.106} C_VEL
LIN {X 0,Y 181.666,Z 226.044,A -85,B 0,C 180,E1 -22904.914,E2 -22904.914} C_VEL
LIN {X 0,Y 184.661,Z 233.797,A -85,B 0,C 180,E1 -22907.028,E2 -22907.028} C_VEL
LIN {X 0,Y 186.658,Z 240.799,A -85,B 0,C 180,E1 -22908.855,E2 -22908.855} C_VEL
LIN {X 0,Y 188.506,Z 251.112,A -85,B 0,C 180,E1 -22911.531,E2 -22911.531} C_VEL
LIN {X 0,Y 189.216,Z 260.788,A -85,B 0,C 180,E1 -22914.161,E2 -22914.161} C_VEL
LIN {X 0,Y 189.016,Z 267.563,A -85,B 0,C 180,E1 -22916.102,E2 -22916.102} C_VEL
LIN {X 0,Y 185.403,Z 276.837,A -85,B 0,C 180,E1 -22918.587,E2 -22918.587} C_VEL
LIN {X 0,Y 181.509,Z 285.81,A -85,B 0,C 180,E1 -22921.686,E2 -22921.686} C_VEL
LIN {X 0,Y 178.617,Z 291.918,A -85,B 0,C 180,E1 -22924.354,E2 -22924.354} C_VEL
LIN {X 0,Y 175.775,Z 297.897,A -85,B 0,C 180,E1 -22927.676,E2 -22927.676} C_VEL
LIN {X 0,Y 173.446,Z 302.62,A -85,B 0,C 180,E1 -22931.085,E2 -22931.085} C_VEL
LIN {X 0,Y 171.535,Z 306.234,A -85,B 0,C 180,E1 -22934.555,E2 -22934.555} C_VEL
LIN {X 0,Y 170.256,Z 308.833,A -85,B 0,C 180,E1 -22938.088,E2 -22938.088} C_VEL
LIN {X 0,Y 169.667,Z 310.054,A -85,B 0,C 180,E1 -22940.462,E2 -22940.462} C_VEL
LIN {X 0,Y 169.266,Z 310.868,A -85,B 0,C 180,E1 -22942.843,E2 -22942.843} C_VEL
LIN {X 0,Y 168.958,Z 311.269,A -85,B 0,C 180,E1 -22947.615,E2 -22947.615} C_VEL
LIN {X 0,Y 169.024,Z 310.903,A -85,B 0,C 180,E1 -22949.998,E2 -22949.998} C_VEL
LIN {X 0,Y 169.194,Z 310.149,A -85,B 0,C 180,E1 -22952.379,E2 -22952.379} C_VEL
LIN {X 0,Y 169.524,Z 308.96,A -85,B 0,C 180,E1 -22954.754,E2 -22954.754} C_VEL
LIN {X 0,Y 170.076,Z 307.196,A -85,B 0,C 180,E1 -22957.36,E2 -22957.36} C_VEL
LIN {X 0,Y 171.073,Z 304.195,A -85,B 0,C 180,E1 -22960.651,E2 -22960.651} C_VEL
LIN {X 0,Y 172.648,Z 299.96,A -85,B 0,C 180,E1 -22964.134,E2 -22964.134} C_VEL
LIN {X 0,Y 175.19,Z 293.544,A -85,B 0,C 180,E1 -22968.111,E2 -22968.111} C_VEL
LIN {X 0,Y 177.991,Z 286.499,A -85,B 0,C 180,E1 -22971.419,E2 -22971.419} C_VEL
LIN {X 0,Y 181.21,Z 277.719,A -85,B 0,C 180,E1 -22974.637,E2 -22974.637} C_VEL
LIN {X 0,Y 184.284,Z 268.715,A -85,B 0,C 180,E1 -22977.231,E2 -22977.231} C_VEL
LIN {X 0,Y 186.109,Z 262.609,A -85,B 0,C 180,E1 -22978.698,E2 -22978.698} C_VEL
LIN {X 0,Y 186.051,Z 255.074,A -85,B 0,C 180,E1 -22980.656,E2 -22980.656} C_VEL
LIN {X 0,Y 185.197,Z 246.259,A -85,B 0,C 180,E1 -22982.787,E2 -22982.787} C_VEL
LIN {X 0,Y 183.121,Z 234.896,A -85,B 0,C 180,E1 -22985.357,E2 -22985.357} C_VEL
LIN {X 0,Y 179.562,Z 223.827,A -85,B 0,C 180,E1 -22987.859,E2 -22987.859} C_VEL
LIN {X 0,Y 175.724,Z 215.618,A -85,B 0,C 180,E1 -22989.845,E2 -22989.845} C_VEL
LIN {X 0,Y 173.627,Z 211.582,A -85,B 0,C 180,E1 -22990.846,E2 -22990.846} C_VEL
LIN {X 0,Y 171.9,Z 208.634,A -85,B 0,C 180,E1 -22991.627,E2 -22991.627} C_VEL
LIN {X 0,Y 171.535,Z 207.238,A -85,B 0,C 180,E1 -22991.904,E2 -22991.904} C_VEL
LIN {X 0,Y 171.376,Z 206.19,A -85,B 0,C 180,E1 -22994.193,E2 -22994.193} C_VEL
LIN {X 0,Y 171.405,Z 206.137,A -85,B 0,C 180,E1 -22999.001,E2 -22999.001} C_VEL
LIN {X 0,Y 171.412,Z 206.132,A -85,B 0,C 180,E1 -23002.047,E2 -23002.047} C_VEL
LIN {X 0,Y 171.395,Z 206.134,A -85,B 0,C 180,E1 -23005.085,E2 -23005.085} C_VEL
LIN {X 0,Y 171.435,Z 206.128,A -85,B 0,C 180,E1 -23010.531,E2 -23010.531} C_VEL
LIN {X 0,Y 171.453,Z 206.107,A -85,B 0,C 180,E1 -23015.8,E2 -23015.8} C_VEL
LIN {X 0,Y 171.596,Z 206.064,A -85,B 0,C 180,E1 -23020.873,E2 -23020.873} C_VEL
LIN {X 0,Y 171.599,Z 206.11,A -85,B 0,C 180,E1 -23025.774,E2 -23025.774} C_VEL
LIN {X 0,Y 171.895,Z 206.063,A -85,B 0,C 180,E1 -23030.587,E2 -23030.587} C_VEL
LIN {X 0,Y 171.803,Z 206.072,A -85,B 0,C 180,E1 -23035.307,E2 -23035.307} C_VEL
LIN {X 0,Y 172.308,Z 206.022,A -85,B 0,C 180,E1 -23039.999,E2 -23039.999} C_VEL
LIN {X 0,Y 171.814,Z 206.082,A -85,B 0,C 180,E1 -23044.692,E2 -23044.692} C_VEL
LIN {X 0,Y 171.87,Z 206.077,A -85,B 0,C 180,E1 -23049.413,E2 -23049.413} C_VEL
LIN {X 0,Y 171.559,Z 206.115,A -85,B 0,C 180,E1 -23054.228,E2 -23054.228} C_VEL
LIN {X 0,Y 171.56,Z 206.117,A -85,B 0,C 180,E1 -23059.592,E2 -23059.592} C_VEL
LIN {X 0,Y 171.455,Z 206.129,A -85,B 0,C 180,E1 -23065.618,E2 -23065.618} C_VEL
LIN {X 0,Y 171.426,Z 206.11,A -85,B 0,C 180,E1 -23070.587,E2 -23070.587} C_VEL
LIN {X 0,Y 171.423,Z 206.251,A -85,B 0,C 180,E1 -23072.903,E2 -23072.903} C_VEL
LIN {X 0,Y 171.883,Z 208.774,A -85,B 0,C 180,E1 -23077.83,E2 -23077.83} C_VEL
LIN {X 0,Y 172.461,Z 212.226,A -85,B 0,C 180,E1 -23083.849,E2 -23083.849} C_VEL
LIN {X 0,Y 172.729,Z 213.925,A -85,B 0,C 180,E1 -23086.536,E2 -23086.536} C_VEL
LIN {X 0,Y 173.851,Z 217.041,A -85,B 0,C 180,E1 -23087.114,E2 -23087.114} C_VEL
LIN {X 0,Y 175.354,Z 219.435,A -85,B 0,C 180,E1 -23087.749,E2 -23087.749} C_VEL
LIN {X 0,Y 179.962,Z 230.389,A -85,B 0,C 180,E1 -23090.141,E2 -23090.141} C_VEL
LIN {X 0,Y 182.096,Z 239.305,A -85,B 0,C 180,E1 -23091.87,E2 -23091.87} C_VEL
LIN {X 0,Y 183.722,Z 251.211,A -85,B 0,C 180,E1 -23094.248,E2 -23094.248} C_VEL
LIN {X 0,Y 184.235,Z 261.113,A -85,B 0,C 180,E1 -23096.413,E2 -23096.413} C_VEL
LIN {X 0,Y 183.854,Z 271.509,A -85,B 0,C 180,E1 -23098.936,E2 -23098.936} C_VEL
LIN {X 0,Y 183.311,Z 277.01,A -85,B 0,C 180,E1 -23100.425,E2 -23100.425} C_VEL
LIN {X 0,Y 179.78,Z 287.037,A -85,B 0,C 180,E1 -23103.288,E2 -23103.288} C_VEL
LIN {X 0,Y 176.719,Z 295.877,A -85,B 0,C 180,E1 -23106.569,E2 -23106.569} C_VEL
LIN {X 0,Y 174.027,Z 302.939,A -85,B 0,C 180,E1 -23109.927,E2 -23109.927} C_VEL
LIN {X 0,Y 171.799,Z 308.582,A -85,B 0,C 180,E1 -23113.363,E2 -23113.363} C_VEL
LIN {X 0,Y 170.343,Z 313.031,A -85,B 0,C 180,E1 -23116.887,E2 -23116.887} C_VEL
LIN {X 0,Y 169.424,Z 316.399,A -85,B 0,C 180,E1 -23120.451,E2 -23120.451} C_VEL
LIN {X 0,Y 169.073,Z 318.076,A -85,B 0,C 180,E1 -23122.838,E2 -23122.838} C_VEL
LIN {X 0,Y 168.852,Z 320.134,A -85,B 0,C 180,E1 -23127.348,E2 -23127.348} C_VEL
LIN {X 0,Y 168.986,Z 320.653,A -85,B 0,C 180,E1 -23130.002,E2 -23130.002} C_VEL
LIN {X 0,Y 168.856,Z 320.662,A -85,B 0,C 180,E1 -23132.681,E2 -23132.681} C_VEL
LIN {X 0,Y 169.074,Z 319.587,A -85,B 0,C 180,E1 -23137.165,E2 -23137.165} C_VEL
LIN {X 0,Y 169.434,Z 318.409,A -85,B 0,C 180,E1 -23139.551,E2 -23139.551} C_VEL
LIN {X 0,Y 170.729,Z 315.173,A -85,B 0,C 180,E1 -23143.891,E2 -23143.891} C_VEL
LIN {X 0,Y 172.64,Z 310.929,A -85,B 0,C 180,E1 -23147.778,E2 -23147.778} C_VEL
LIN {X 0,Y 175.028,Z 305.927,A -85,B 0,C 180,E1 -23151.185,E2 -23151.185} C_VEL
LIN {X 0,Y 176.612,Z 302.739,A -85,B 0,C 180,E1 -23152.959,E2 -23152.959} C_VEL
LIN {X 0,Y 177.492,Z 299.658,A -85,B 0,C 180,E1 -23154.56,E2 -23154.56} C_VEL
LIN {X 0,Y 177.286,Z 294.305,A -85,B 0,C 180,E1 -23157.261,E2 -23157.261} C_VEL
LIN {X 0,Y 177.269,Z 288.415,A -85,B 0,C 180,E1 -23159.839,E2 -23159.839} C_VEL
LIN {X 0,Y 178.393,Z 284.443,A -85,B 0,C 180,E1 -23161.198,E2 -23161.198} C_VEL
LIN {X 0,Y 179.961,Z 280.108,A -85,B 0,C 180,E1 -23162.477,E2 -23162.477} C_VEL
LIN {X 0,Y 181.03,Z 270.267,A -85,B 0,C 180,E1 -23165.386,E2 -23165.386} C_VEL
LIN {X 0,Y 181.117,Z 260.569,A -85,B 0,C 180,E1 -23167.984,E2 -23167.984} C_VEL
LIN {X 0,Y 180.539,Z 251.039,A -85,B 0,C 180,E1 -23170.323,E2 -23170.323} C_VEL
LIN {X 0,Y 179.21,Z 243.202,A -85,B 0,C 180,E1 -23172.251,E2 -23172.251} C_VEL
LIN {X 0,Y 177.52,Z 237.64,A -85,B 0,C 180,E1 -23173.738,E2 -23173.738} C_VEL
LIN {X 0,Y 173.414,Z 228.281,A -85,B 0,C 180,E1 -23176.525,E2 -23176.525} C_VEL
LIN {X 0,Y 171.032,Z 223.601,A -85,B 0,C 180,E1 -23178.015,E2 -23178.015} C_VEL
LIN {X 0,Y 169.13,Z 220.151,A -85,B 0,C 180,E1 -23179.18,E2 -23179.18} C_VEL
LIN {X 0,Y 168.271,Z 218.616,A -85,B 0,C 180,E1 -23179.69,E2 -23179.69} C_VEL
LIN {X 0,Y 166.251,Z 215.747,A -85,B 0,C 180,E1 -23180.843,E2 -23180.843} C_VEL
LIN {X 0,Y 165.372,Z 213.158,A -85,B 0,C 180,E1 -23181.572,E2 -23181.572} C_VEL
LIN {X 0,Y 164.976,Z 210.811,A -85,B 0,C 180,E1 -23186.372,E2 -23186.372} C_VEL
LIN {X 0,Y 164.868,Z 209.545,A -85,B 0,C 180,E1 -23189.234,E2 -23189.234} C_VEL
LIN {X 0,Y 164.47,Z 207.414,A -85,B 0,C 180,E1 -23194.703,E2 -23194.703} C_VEL
LIN {X 0,Y 164.389,Z 207.007,A -85,B 0,C 180,E1 -23197.371,E2 -23197.371} C_VEL
LIN {X 0,Y 164.515,Z 206.994,A -85,B 0,C 180,E1 -23200.017,E2 -23200.017} C_VEL
LIN {X 0,Y 164.522,Z 206.99,A -85,B 0,C 180,E1 -23205.15,E2 -23205.15} C_VEL
LIN {X 0,Y 164.759,Z 206.96,A -85,B 0,C 180,E1 -23210.176,E2 -23210.176} C_VEL
LIN {X 0,Y 164.821,Z 206.952,A -85,B 0,C 180,E1 -23212.651,E2 -23212.651} C_VEL
LIN {X 0,Y 165.035,Z 206.925,A -85,B 0,C 180,E1 -23217.56,E2 -23217.56} C_VEL
LIN {X 0,Y 165.279,Z 206.896,A -85,B 0,C 180,E1 -23220.001,E2 -23220.001} C_VEL
LIN {X 0,Y 164.763,Z 206.962,A -85,B 0,C 180,E1 -23224.894,E2 -23224.894} C_VEL
LIN {X 0,Y 164.819,Z 206.954,A -85,B 0,C 180,E1 -23227.35,E2 -23227.35} C_VEL
LIN {X 0,Y 164.695,Z 206.97,A -85,B 0,C 180,E1 -23231.059,E2 -23231.059} C_VEL
LIN {X 0,Y 164.473,Z 206.996,A -85,B 0,C 180,E1 -23237.405,E2 -23237.405} C_VEL
LIN {X 0,Y 164.468,Z 206.997,A -85,B 0,C 180,E1 -23239.991,E2 -23239.991} C_VEL
LIN {X 0,Y 164.381,Z 207.008,A -85,B 0,C 180,E1 -23246.129,E2 -23246.129} C_VEL
LIN {X 0,Y 164.369,Z 207.012,A -85,B 0,C 180,E1 -23251.228,E2 -23251.228} C_VEL
LIN {X 0,Y 164.325,Z 207.117,A -85,B 0,C 180,E1 -23253.78,E2 -23253.78} C_VEL
LIN {X 0,Y 164.438,Z 207.951,A -85,B 0,C 180,E1 -23256.169,E2 -23256.169} C_VEL
LIN {X 0,Y 165.628,Z 210.871,A -85,B 0,C 180,E1 -23257.015,E2 -23257.015} C_VEL
LIN {X 0,Y 167.92,Z 213.709,A -85,B 0,C 180,E1 -23258.313,E2 -23258.313} C_VEL
LIN {X 0,Y 169.943,Z 217.431,A -85,B 0,C 180,E1 -23259.609,E2 -23259.609} C_VEL
LIN {X 0,Y 171.191,Z 219.431,A -85,B 0,C 180,E1 -23260.35,E2 -23260.35} C_VEL
LIN {X 0,Y 173.608,Z 224.018,A -85,B 0,C 180,E1 -23261.91,E2 -23261.91} C_VEL
LIN {X 0,Y 177.389,Z 231.993,A -85,B 0,C 180,E1 -23264.511,E2 -23264.511} C_VEL
LIN {X 0,Y 180.128,Z 240.149,A -85,B 0,C 180,E1 -23266.892,E2 -23266.892} C_VEL
LIN {X 0,Y 182.033,Z 250.022,A -85,B 0,C 180,E1 -23269.622,E2 -23269.622} C_VEL
LIN {X 0,Y 182.916,Z 259.633,A -85,B 0,C 180,E1 -23272.372,E2 -23272.372} C_VEL
LIN {X 0,Y 182.862,Z 267.609,A -85,B 0,C 180,E1 -23274.796,E2 -23274.796} C_VEL
LIN {X 0,Y 181.589,Z 271.556,A -85,B 0,C 180,E1 -23275.863,E2 -23275.863} C_VEL
LIN {X 0,Y 177.953,Z 280.162,A -85,B 0,C 180,E1 -23278.448,E2 -23278.448} C_VEL
LIN {X 0,Y 173.998,Z 288.499,A -85,B 0,C 180,E1 -23281.667,E2 -23281.667} C_VEL
LIN {X 0,Y 170.646,Z 295.108,A -85,B 0,C 180,E1 -23284.969,E2 -23284.969} C_VEL
LIN {X 0,Y 167.524,Z 301.341,A -85,B 0,C 180,E1 -23289.109,E2 -23289.109} C_VEL
LIN {X 0,Y 165.23,Z 305.327,A -85,B 0,C 180,E1 -23292.678,E2 -23292.678} C_VEL
LIN {X 0,Y 164.175,Z 307.378,A -85,B 0,C 180,E1 -23295.116,E2 -23295.116} C_VEL
LIN {X 0,Y 162.663,Z 310.232,A -85,B 0,C 180,E1 -23300.047,E2 -23300.047} C_VEL
